(* CoDeSys 2.3.9.48 project: 4.2_EOT20170112.pro *)
(* Libraries: SYSLIBMEM.LIB 8.11.10 18:37:48, C:\Program Files (x86)\WAGO Software\CoDeSys V2.3\Targets\WAGO\Libraries\Application\WagoLibMBX_System_01.lib 22.10.13 22:28:54, C:\Program Files (x86)\WAGO Software\CoDeSys V2.3\Targets\WAGO\Libraries\Application\WagoLibMBX_01.lib 20.3.12 22:32:38, C:\Program Files (x86)\WAGO Software\CoDeSys V2.3\Targets\WAGO\Libraries\Application\WagoLib_CAN_Gateway_02.lib 25.11.15 18:32:40, Util.lib 26.9.14 10:12:46, Standard.lib 8.11.10 18:37:48, SYSLIBCALLBACK.LIB 8.11.10 18:37:48, WagoLibModbus_IP_01.lib 12.2.16 17:20:24, SysLibSockets.lib 5.5.11 15:22:24, WagoLibSockets.lib 14.5.12 18:49:54, NETVARUDP_LIB_V23.LIB 8.11.10 18:37:48, Wago_MBCFG_ETHERNET_01.lib 1.4.15 20:24:28, Wago_MBCFG_COMMON_01.lib 1.4.15 20:24:28 *)

(* PLC configuration (modules and I/O channels)
0753-0430 8 DI 24 V DC 3.0ms [Type_1_8_Channels] node 0, in %IB12 out %QB24 {INTTypePAAssignment = PLC; INTTypeModule = plugged}
  AT %IX6.0 [BOOLOnX_I] Ch_1 Digital input
  AT %IX6.1 [BOOLOnX_I] Ch_2 Digital input
  AT %IX6.2 [BOOLOnX_I] Ch_3 Digital input
  AT %IX6.3 [BOOLOnX_I] Ch_4 Digital input
  AT %IX6.4 [BOOLOnX_I] Ch_5 Digital input
  AT %IX6.5 [BOOLOnX_I] Ch_6 Digital input
  AT %IX6.6 [BOOLOnX_I] Ch_7 Digital input
  AT %IX6.7 [BOOLOnX_I] Ch_8 Digital input
0753-0430 8 DI 24 V DC 3.0ms [Type_1_8_Channels] node 1, in %IB12 out %QB24 {INTTypePAAssignment = PLC; INTTypeModule = plugged}
  AT %IX6.8 [BOOLOnX_I] Ch_1 Digital input
  AT %IX6.9 [BOOLOnX_I] Ch_2 Digital input
  AT %IX6.10 [BOOLOnX_I] Ch_3 Digital input
  AT %IX6.11 [BOOLOnX_I] Ch_4 Digital input
  AT %IX6.12 [BOOLOnX_I] Ch_5 Digital input
  AT %IX6.13 [BOOLOnX_I] Ch_6 Digital input
  AT %IX6.14 [BOOLOnX_I] Ch_7 Digital input
  AT %IX6.15 [BOOLOnX_I] Ch_8 Digital input
0753-0430 8 DI 24 V DC 3.0ms [Type_1_8_Channels] node 2, in %IB13 out %QB24 {INTTypePAAssignment = PLC; INTTypeModule = plugged}
  AT %IX7.0 [BOOLOnX_I] Ch_1 Digital input
  AT %IX7.1 [BOOLOnX_I] Ch_2 Digital input
  AT %IX7.2 [BOOLOnX_I] Ch_3 Digital input
  AT %IX7.3 [BOOLOnX_I] Ch_4 Digital input
  AT %IX7.4 [BOOLOnX_I] Ch_5 Digital input
  AT %IX7.5 [BOOLOnX_I] Ch_6 Digital input
  AT %IX7.6 [BOOLOnX_I] Ch_7 Digital input
  AT %IX7.7 [BOOLOnX_I] Ch_8 Digital input
AT %QX12.0 [BOOLOnX_Q] Ch_1 Digital output
AT %QX12.1 [BOOLOnX_Q] Ch_2 Digital output
AT %QX12.2 [BOOLOnX_Q] Ch_3 Digital output
AT %QX12.3 [BOOLOnX_Q] Ch_4 Digital output
AT %QX12.4 [BOOLOnX_Q] Ch_5 Digital output
AT %QX12.5 [BOOLOnX_Q] Ch_6 Digital output
AT %QX12.6 [BOOLOnX_Q] Ch_7 Digital output
AT %QX12.7 [BOOLOnX_Q] Ch_8 Digital output
AT %QX12.8 [BOOLOnX_Q] Ch_1 Digital output
AT %QX12.9 [BOOLOnX_Q] Ch_2 Digital output
AT %QX12.10 [BOOLOnX_Q] Ch_3 Digital output
AT %QX12.11 [BOOLOnX_Q] Ch_4 Digital output
AT %QX12.12 [BOOLOnX_Q] Ch_5 Digital output
AT %QX12.13 [BOOLOnX_Q] Ch_6 Digital output
AT %QX12.14 [BOOLOnX_Q] Ch_7 Digital output
AT %QX12.15 [BOOLOnX_Q] Ch_8 Digital output
AT %QX13.0 [BOOLOnX_Q] Ch_1 Digital output
AT %QX13.1 [BOOLOnX_Q] Ch_2 Digital output
AT %QX13.2 [BOOLOnX_Q] Ch_3 Digital output
AT %QX13.3 [BOOLOnX_Q] Ch_4 Digital output
AT %QX13.4 [BOOLOnX_Q] Ch_5 Digital output
AT %QX13.5 [BOOLOnX_Q] Ch_6 Digital output
AT %QX13.6 [BOOLOnX_Q] Ch_7 Digital output
AT %QX13.7 [BOOLOnX_Q] Ch_8 Digital output
AT %QW0 [WORDOnW_Q] Ch_1 Analog output
AT %QW1 [WORDOnW_Q] Ch_2 Analog output
AT %QW2 [WORDOnW_Q] Ch_3 Analog output
AT %QW3 [WORDOnW_Q] Ch_4 Analog output
AT %QW4 [WORDOnW_Q] Ch_1 Analog output
AT %QW5 [WORDOnW_Q] Ch_2 Analog output
AT %QW6 [WORDOnW_Q] Ch_3 Analog output
AT %QW7 [WORDOnW_Q] Ch_4 Analog output
AT %IW0 [WORDOnW_I] Ch_1 Input word
AT %IW1 [WORDOnW_I] Ch_2 Input word
AT %IW2 [WORDOnW_I] Ch_1 Input word
AT %IW3 [WORDOnW_I] Ch_2 Input word
AT %IW4 [WORDOnW_I] Ch_1 Input word
AT %IW5 [WORDOnW_I] Ch_2 Input word
0753-0555 4 AO 4-20mA [Type_14_4_Channels] node 6, in %IB20 out %QB32 {INTTypePAAssignment = PLC; INTTypeModule = plugged}
  AT %QW8 [WORDOnW_Q] Ch_1 Analog output
  AT %QW9 [WORDOnW_Q] Ch_2 Analog output
  AT %QW10 [WORDOnW_Q] Ch_3 Analog output
  AT %QW11 [WORDOnW_Q] Ch_4 Analog output
Fieldbus variables [FB_VARS] node 1, in %IB0 out %QB0
Flag variables [FLAG_VARS] node 2, in %IB0 out %QB0
Modbus-Master [MB_MASTER] node 3, in %IB0 out %QB0
*)

(* Global variable list: Global_Variables *)
VAR_GLOBAL

	(*---------------------Control transfer between WING EOT and BRG CENR EOT---------------------*)
	(*control flag*)
	(*control in bridge*)
	BRG_IN_CONTROL_P: BOOL;

	BRG_CENR_IN_CONTROL: BOOL := TRUE;
	BRG_PORT_IN_CONTROL: BOOL := FALSE;
	BRG_STBD_IN_CONTROL: BOOL := FALSE;

	(*during control transfer process flag*)
	CONTROL_TRANS_PROCESS_FLAG: BOOL := FALSE;

	(*EOT LAMP*)
	BRIDGE_PORT_EOT_IN_CONTROL_LAMP: BOOL;
	BRIDGE_STBD_EOT_IN_CONTROL_LAMP: BOOL;
	PORT_EOT_IN_CONTROL_LAMP: BOOL;
	STBD_EOT_IN_CONTROL_LAMP: BOOL;

	(*EOT MVL*)
	PORT_WING_EOT_MVL: WORD;
	CENT_EOT_MVL: WORD;
	STBD_WING_EOT_MVL: WORD;

	(*BUZZER EOT*)
	BRIDGE_BUZZER: BOOL;
	PORT_BUZZER: BOOL;
	STBD_BUZZER: BOOL;


	(*TAKE and SUPPLY button*)
	(*CNTR BUTTON*)
	PORT_BUTTON_EOT_IN_CNTR: BOOL;
	STBD_BUTTON_EOT_IN_CNTR: BOOL;
	(*STBD,PORT  BUTTON*)
	STBD_BUTTON_EOT: BOOL;
	PORT_BUTTON_EOT: BOOL;

	(*Flasher_frequency*)
	Flasher_frequency_P: REAL;


	(*---------------------4.1.7.1.1  MVL Command--------------------*)
	(*input*)
	TELEGRAPH_POSITION_BR: WORD;
	TELEGRAPH_POSITION_CR: WORD;
	TELEGRAPH_POSITION_LC: WORD;

	ECR_AUT_CTRL: BOOL;
	LOCAL_MAN_CTRL: BOOL;
	(*output*)
	TELEGRAPH_INDICATOR_BR: WORD;
	TELEGRAPH_INDICATOR_BR_PORT: WORD;
	TELEGRAPH_INDICATOR_BR_STBD: WORD;
	TELEGRAPH_INDICATOR_ECR: WORD;
	TELEGRAPH_INDICATOR_LC: WORD;

	(**************MVL POWER LOST**************)
	(*INPUT*)
	ECR_TElegraph_POWER_LOST_P: BOOL;
	LOCAL_TElegraph_POWER_LOST_P: BOOL;
	PORT_TElegraph_POWER_LOST_P: BOOL;
	STBD_TElegraph_POWER_LOST_P: BOOL;
	BR_TElegraph_POWER_LOST_P: BOOL;

	TELEGRAPH_SUB_SYS_PWR_LOST: BOOL;



	(*---------------------4.1.7.1.2  Sub-telegraph function--------------------*)
	(*current status
	0 = NOSTATUS; 1 = STANDBY; 2 = AT SEA; 3 = FWE*)
	AUX_EOT_STATUS: UDINT := 0;

	(*PUSHBUTTON*)
	PUSHBUTTON_STANDBY_BRG: BOOL;
	PUSHBUTTON_ATSEA_BRG: BOOL;
	PUSHBUTTON_FWE_BRG: BOOL;

	PUSHBUTTON_STANDBY_MCR: BOOL;
	PUSHBUTTON_ATSEA_MCR: BOOL;
	PUSHBUTTON_FWE_MCR: BOOL;

	(*indicator*)
	INDICATOR_STANDBY_BRG: BOOL;
	INDICATOR_ATSEA_BRG: BOOL;
	INDICATOR_FWE_BRG: BOOL;

	INDICATOR_STANDBY_MCR: BOOL;
	INDICATOR_ATSEA_MCR: BOOL;
	INDICATOR_FWE_MCR: BOOL;

	INDICATOR_STANDBY_LC: BOOL;
	INDICATOR_ATSEA_LC: BOOL;
	INDICATOR_FWE_LC: BOOL;

	(*buzzers, FALSE = silence; TRUE = activated*)
	BUZZER_BRG: BOOL;
	BUZZER_MCR: BOOL;

	(*Is during switch process NO = FALSE; YES = TRUE*)
	MODE_TRANSFER_FLAG: BOOL := FALSE;

	H_AT_SEA: BOOL; (*PROEOT0003*)
	H_STAND_BY: BOOL;(*PROEOT0004*)
	H_FINSHED_WITH_ENGINE: BOOL;(*PROEOT0005*)


	(*---------------------4.1.7.1.3  Wrong way--------------------*)
	(*input*)
	MVL_POSITION_AHEAD: BOOL;
	MVL_POSITION_ASTERN: BOOL;
	ENGINE_TURN_AHEAD: BOOL;
	ENGINE_TURN_ASTERN: BOOL;
	MCR_LC_CONTROL: BOOL;
	ECR_MAN_CONTROL: BOOL;

	(*output*)
	WRONG_WAY: BOOL;

	(*---------------------4.1.7.1.4  Mismatch Alarm--------------------*)
	(*input*)
	TELEGRAPH_ORDER_THRESHOLD_INPUT: WORD;(*2ma*)
	(*output*)
	TELEGRAPH_ORDER_BR: BOOL;
	TELEGRAPH_ORDER_PORT: BOOL;
	TELEGRAPH_ORDER_STBD: BOOL;
	TELEGRAPH_ORDER_ECR: BOOL;
	TELEGRAPH_ORDER_LC: BOOL;

	TELEGRAPH_COINCIDENCE: BOOL;

	(*silence  MISMATCH BUZZER*)
	ESS_BR_ALARM_ACK_P:    BOOL;
	ESS_ECR_ALARM_ACK_P:   BOOL;
	ESS_PORT_ALARM_ACK_P:   BOOL;
	ESS_STBD_ALARM_ACK_P:   BOOL;

	(*---------------------4.1.7.1.5  EOT system failure Alarm--------------------*)
	(*input*)
	PASSIVE_FAIL_THRESHOLD: WORD;(*2ma*)
	(*output*)
	PASSIVE_FAILURE_BR: BOOL;
	PASSIVE_FAILURE_BR_PORT: BOOL;
	PASSIVE_FAILURE_BR_STBD: BOOL;
	PASSIVE_FAILURE_ECR: BOOL;
	PASSIVE_FAILURE_LC: BOOL;

	TELEGRAPH_SYSTEM_FAIL_XS9021A: BOOL;

	(*---------------------LAMP TEST PB FROM RCS--------------------*)
	ECR_LAMP_TEST_PB: BOOL;
	BR_LAMP_TEST_PB: BOOL;
	PORT_LAMP_TEST_PB: BOOL;
	STBD_LAMP_TEST_PB: BOOL;

	(*4 lamp test PB OR*)
	LAMP_TEST_PB:	BOOL;
	BRIDGE_LAMP_TEST_PB:	BOOL;

	(*-------------------------------AMPERE STAGE TO HMI-------------------------------*)
	(*750-452  AI 输入模块 0~20mA, 20mA对应32760,  AD_Scale 为32760/20*)
	AD_Scale: WORD := 1638;
	(*750-555  AO 输出模块 4~20mA, 20mA对应32760, DA_Scale 为32760/16*)
	DA_Scale: WORD := 2048;

	AMPERE_STAGE_TO_HMI: WORD;		(*
												   bit 0	Emergency  AS
												   bit 1   FULL.AS
												   bit 2   HALF AS
												   bit 3  	SLOW  AS
												   bit 4   DEAD  S. AH
												   bit 5   STOP
												   bit 6   DEAD  S. AH
												   bit 7   SLOW  AH
												   bit 8   HALF  AH
												   bit 9   FULL  AH 
												   bit 10   Full SEA  AH*)


	(*LEVEL	INDICATOR*)
	Telegraph_Indicator_Full_SEA_AH: BOOL;
	Telegraph_Indicator_FULL_AH: BOOL;
	Telegraph_Indicator_HALF_AH: BOOL;
	Telegraph_Indicator_SLOW_AH: BOOL;
	Telegraph_Indicator_DEAD_S_AH: BOOL;
	Telegraph_Indicator_STOP: BOOL;
	Telegraph_Indicator_DEAD_S_AS: BOOL;
	Telegraph_Indicator_SLOW_AS: BOOL;
	Telegraph_Indicator_HALF_AS: BOOL;
	Telegraph_Indicator_FULL_AS: BOOL;
	Telegraph_Indicator_Emergency_AS: BOOL;

	(*LEVEL CMD*)
	Telegraph_CMD_Full_SEA_AH: BOOL;
	Telegraph_CMD_FULL_AH: BOOL;
	Telegraph_CMD_HALF_AH: BOOL;
	Telegraph_CMD_SLOW_AH: BOOL;
	Telegraph_CMD_DEAD_S_AH: BOOL;
	Telegraph_CMD_STOP: BOOL;
	Telegraph_CMD_DEAD_S_AS: BOOL;
	Telegraph_CMD_SLOW_AS: BOOL;
	Telegraph_CMD_HALF_AS: BOOL;
	Telegraph_CMD_FULL_AS: BOOL;
	Telegraph_CMD_Emergency_AS: BOOL;

	(***************************MVL_COMMD_TO_AO*******************************)
	BR_MVL_COMMD_TO_RCS_P: WORD;
	ECR_MVL_COMMD_TO_RCS_P: WORD;

	(*INDICATOR OF  BR  MCR  LC*)
	BR_Indicator_Position_Pointer_P:	WORD;
	ECR_Indicator_Position_Pointer_P:  WORD;
	LOCAL_Indicator_Position_Pointer_P:	WORD;

	BR_PORT_Indicator_Position_Pointer_P:	WORD;
	BR_STBD_Indicator_Position_Pointer_P:	WORD;

	(*TEST*)
	TEST_LOCAL_Telegraph_Position_Pointer_P :  WORD;

	(****************************MVL_TO_RCS_TEST_MBS---12.27*******************************)
	BR_MVL_TO_RCS_MBS_P	AT %QW275:	WORD;
	ECR_MVL_TO_RCS_MBS_P		AT %QW277:	WORD;

	BR_MVL_TO_RCS_MBS_P1		AT %QW279:	WORD;
	ECR_MVL_TO_RCS_MBS_P1		AT %QW281:	WORD;


	(***************************EOT HW Signal list*******************************)
	(*-----------AI----------*)
	BR_MVL_COMMD									AT	%IW0: WORD;(*PROEOT1001*)
	ECR_MVL_COMMD								AT	%IW1: WORD;(*PROEOT1002*)
	LOCAL_MVL_COMMD							AT	%IW2: WORD;(*PROEOT1003*)
	PORT_BR_MVL_COMMD: 				WORD;(*PROEOT1004*)
	STBD_BR_MVL_COMMD: 				WORD;(*PROEOT1005*)

	(*-----------AO----------*)
	BR_Indicator_Position_Pointer					AT	%QW0: WORD;(*PROEOT1006*)
	BR_MVL_COMMD_TO_RCS					       AT %QW4: WORD;(*PROEOT1007*)
	ECR_Indicator_Position_Pointer					AT	%QW1: WORD;(*PROEOT1008*)
	ECR_MVL_COMMD_TO_RCS 					AT%QW5: WORD;(*PROEOT1009*)
	LOCAL_Indicator_Position_Pointer				AT	%QW2: WORD;(*PROEOT1010*)
	PORT_BR_Indicator_Position_Pointer: REAL;(*PROEOT1011*)
	STBD_BR_Indicator_Position_Pointer: REAL;(*PROEOT1012*)
	(*TEST*)
	TEST_LOCAL_Telegraph_Position_Pointer		AT	%QW3: WORD;(*PROEOT1010*)

	(*-----------DI----------*)
	STANDBY_BR_PB								AT	%IX6.0: BOOL;(*PROEOT1013*)
	AT_SEA_BR_PB									AT	%IX6.1: BOOL;(*PROEOT1014*)
	FWE_BR_PB										AT	%IX6.2: BOOL;(*PROEOT1015*)
	BR_TElegraph_POWER_LOST					AT	%IX6.3: BOOL;(*PROEOT1016*)
	STANDBY_ECR_AUT_PB						AT	%IX6.4: BOOL;(*PROEOT1017*)
	AT_SEA_ECR_AUT_PB							AT	%IX6.5: BOOL;(*PROEOT1018*)
	FWE_ECR_AUT_PB								AT	%IX6.6: BOOL;(*PROEOT1019*)
	ECR_TElegraph_POWER_LOST				AT	%IX6.7: BOOL;(*PROEOT1020*)
	LOCAL_TElegraph_POWER_LOST				AT	%IX6.10: BOOL;(*PROEOT1021*)
	PORT_TElegraph_POWER_LOST: BOOL;(*PROEOT1022*)
	STBD_TElegraph_POWER_LOST: BOOL;(*PROEOT1023*)
	BR_CENTRL_PORT_APPLY_FOR_CONTROL: BOOL;(*PROEOT1024*)
	BR_CENTRL_STBD_APPLY_FOR_CONTROL: BOOL;(*PROEOT1025*)
	BR_PORT_APPLY_FOR_CONTROL: BOOL;(*PROEOT1026*)
	BR_STBD_APPLY_FOR_CONTROL: BOOL;(*PROEOT1027*)
	LOCAL_IN_CONTROL_TAKE_ON				AT	%IX7.1: BOOL;(*PROEOT1028*)


	(*-----------DO----------*)
	STANDBY_BR_INDICATOR									AT	%QX12.0: BOOL;(*PROEOT1029*)
	AT_SEA_BR_PB_INDICATOR								AT	%QX12.1: BOOL;(*PROEOT1030*)
	FWE_BR_PB_INDICATOR									AT	%QX12.2: BOOL;(*PROEOT1031*)
	BR_TELEGRAPH_ORDER_Acoustic_Signal				AT	%QX12.3: BOOL;(*PROEOT1032*)
	STANDBY_ECR_AUT_PB_INDICATOR						AT	%QX12.4: BOOL;(*PROEOT1033*)
	AT_SEA_ECR_AUT_PB_INDICATOR						AT	%QX12.5: BOOL;(*PROEOT1034*)
	FWE_ECR_AUT_PB_INDICATOR							AT	%QX12.6: BOOL;(*PROEOT1035*)
	ECR_TELEGRAPH_ORDER_Acoustic_Signal				AT	%QX12.7: BOOL;(*PROEOT1036*)
	STANDBY_LOCAL_INDICATOR: BOOL;(*PROEOT1037*)
	AT_SEA_LOCAL_INDICATOR: BOOL;(*PROEOT1038*)
	FWE_LOCAL_INDICATOR: BOOL;(*PROEOT1039*)
	LOCAL_TELEGRAPH_ORDER_Acoustic_Signal			AT	%QX12.10: BOOL;(*PROEOT1040*)
	PORT_TELEGRAPH_ORDER_Acoustic_Signal: BOOL;(*PROEOT1041*)
	STBD_TELEGRAPH_ORDER_Acoustic_Signal: BOOL;(*PROEOT1042*)
	BR_CENTRL_PORT_CONTROL_IN_CONTROL: BOOL;(*PROEOT1043*)
	BR_CENTRL_STBD_CONTROL_IN_CONTROL: BOOL;(*PROEOT1044*)
	BR_PORT_CONTROL_IN_CONTROL: BOOL;(*PROEOT1045*)
	BR_STBD_CONTROL_IN_CONTROL: BOOL;(*PROEOT1046*)
	LOCAL_IN_CONTROL_TAKE_ON_INDICATOR				AT	%QX13.1: BOOL;(*PROEOT1047*)
	Telegraph_System_Failure_ALM								AT	%QX13.2: BOOL;(*PROEOTXS9021A*)
	HW_WRONG_WAY_BR										AT	%QX13.3:  BOOL;
	HW_WRONG_WAY_ECR										AT	%QX13.4:  BOOL;
	HW_WRONG_WAY_LC										AT	%QX13.5:  BOOL;

	(*PORT or STBD in control *)
	HW_PORT_IN_CONTROL: BOOL;	(*PROEOT1048*)
	HW_STBD_IN_CONTROL: BOOL;	(*PROEOT1049*)


	(****************************EOT & HMI COMMUNICATION SIGNALS LIST*******************************)
	(*STRING*)

  	SWD_swd_ctr_mode_0 AT %QW271: UINT;


	(*SDO*)

	LOCAL_MAN_TAKE_OVER   AT	%QX260.11: BOOL;(*PROEOT0019       SP_swd_perm_eot1_12_62*)
	H_PORT_WING_CONTRL  AT	%QX260.12: BOOL;(*PROEOT0025       SP_swd_perm_eot1_13_62*)
	H_STBD_WING_CONTRL   AT	%QX259.13: BOOL;(*PROEOT0026    SP_swd_perm_eot1_14_62*)

	H_BR_TElegraph_POWER_LOST  AT	%QX261.0: BOOL;(*PROEOT0029    SP_swd_perm_eot2_1_62*)
	H_ECR_TElegraph_POWER_LOST  AT	%QX261.1: BOOL;(*PROEOT0030   SP_swd_perm_eot2_2_62*)
	H_LOCAL_TElegraph_POWER_LOST  AT	%QX261.2: BOOL;(*PROEOT0031   SP_swd_perm_eot2_3_62*)
	H_PORT_TElegraph_POWER_LOST  AT	%QX261.3: BOOL;(*PROEOT0032    SP_swd_perm_eot2_4_62*)
	H_STBD_TElegraph_POWER_LOST  AT	%QX261.4: BOOL;(*PROEOT0033   SP_swd_perm_eot2_5_62*)

	H_BR_TElegraph_PASSIVE_FAIL  AT	%QX261.5: BOOL;(*PROEOT0034  SP_swd_perm_eot2_6_62*)
	H_ECR_TElegraph_PASSIVE_FAIL  AT	%QX261.6: BOOL;(*PROEOT0035   SP_swd_perm_eot2_7_62*)
	H_LOCAL_TElegraph_PASSIVE_FAIL  AT	%QX261.7: BOOL;(*PROEOT0036   SP_swd_perm_eot2_8_62*)
	H_PORT_TElegraph_PASSIVE_FAIL  AT	%QX261.8: BOOL;(*PROEOT0037    SP_swd_perm_eot2_9_62*)
	H_STBD_TElegraph_PASSIVE_FAIL  AT	%QX261.9: BOOL;(*PROEOT0038   SP_swd_perm_eot2_10_62*)

	TELEGRAPH_HORN_ALARM_MBO   AT   %QX261.10: BOOL;   (*PROEOT0039   SP_swd_perm_eot2_11_62*)
	TELEGRAPH_SUB_SYS_PWR_LOST_MBO   AT   %QX261.11: BOOL;   (*PROEOT0044   SP_swd_perm_eot2_12_62*)
	TELEGRAPH_SYS_PASS_FAIL_9021A_MBO   AT   %QX261.12: BOOL;  (*PROEOTXS9021A   SP_swd_perm_eot2_13_62*)

	H_TELEGRAPH_COINCIDENCE   AT   %QX261.13: BOOL;  (*PROEOT9001  SP_swd_perm_eot2_14_62*)
	H_WRONG_WAY	 AT   %QX261.14:  BOOL; 	(*PROEOT9050  SP_swd_perm_eot2_15_62*)

	(*Corresponding  Ampere to  HMI-----------------------New Signal*)
	Telegraph_Indicator_Full_SEA_AH_MBO      AT  %QX260.0: BOOL;  (*PROEOT0001      SP_swd_perm_eot1_1_62 *)
	Telegraph_Indicator_FULL_AH_MBO      AT  %QX260.1: BOOL;  (*PROEOT0002      SP_swd_perm_eot1_2_62 *)
	Telegraph_Indicator_HALF_AH_MBO      AT  %QX260.2: BOOL;  (*PROEOT0003      SP_swd_perm_eot1_3_62 *)
	Telegraph_Indicator_SLOW_AH_MBO      AT  %QX260.3: BOOL;  (*PROEOT0004      SP_swd_perm_eot1_4_62 *)
	Telegraph_Indicator_DEAD_S_AH_MBO      AT  %QX260.4: BOOL;  (*PROEOT0005      SP_swd_perm_eot1_5_62 *)
	Telegraph_Indicator_STOP_MBO      AT  %QX260.5: BOOL;  (*PROEOT0006      SP_swd_perm_eot1_6_62 *)
	Telegraph_Indicator_DEAD_S_AS_MBO      AT  %QX260.6: BOOL;  (*PROEOT0007      SP_swd_perm_eot1_7_62 *)
	Telegraph_Indicator_SLOW_AS_MBO      AT  %QX260.7: BOOL;  (*PROEOT0008      SP_swd_perm_eot1_8_62 *)
	Telegraph_Indicator_HALF_AS_MBO      AT  %QX260.8: BOOL;  (*PROEOT0009      SP_swd_perm_eot1_9_62 *)
	Telegraph_Indicator_FULL_AS_MBO      AT  %QX260.9: BOOL;  (*PROEOT0010      SP_swd_perm_eot1_10_62 *)
	Telegraph_Indicator_Emergency_AS_MBO      AT  %QX260.10: BOOL;  (*PROEOT0011      SP_swd_perm_eot1_11_62 *)


	(****************************RCS TO EOT 		ESS TO EOT   MODBUS  COMMUNICATION SIGNALS LIST*******************************)
(*	FRM_BR_CONTROL     AT  %IX262.0: BOOL;    (*PROEOT0017      SP_swd_perm_eotout_1_62  *)
	FRM_ECR_AUT_CONTROL     AT  %IX262.1: BOOL;    (*PROEOT0018      SP_swd_perm_eotout_2_62  *)
	FRM_ECR_LAMP_TEST_PB     AT  %IX262.2: BOOL;    (*PROEOT0040      SP_swd_perm_eotout_3_62  *)
	FRM_BR_LAMP_TEST_PB     AT  %IX262.3: BOOL;    (*PROEOT0041      SP_swd_perm_eotout_4_62  *)
	FRM_PORT_LAMP_TEST_PB     AT  %IX262.4: BOOL;    (*PROEOT0042      SP_swd_perm_eotout_5_62  *)
	FRM_STBD_LAMP_TEST_PB     AT  %IX262.5: BOOL;    (*PROEOT0043      SP_swd_perm_eotout_6_62  *)


	ESS_BR_ALARM_ACK     AT  %IX262.6: BOOL;    (*PROEOT0045	SP_swd_perm_eotout_7_62  *)
	ESS_ECR_ALARM_ACK     AT  %IX262.7: BOOL;    (*PROEOT0046	SP_swd_perm_eotout_8_62  *)
	ESS_PORT_ALARM_ACK     AT  %IX262.8: BOOL;    (*PROEOT0047	SP_swd_perm_eotout_9_62  *)
	ESS_STBD_ALARM_ACK     AT  %IX262.9: BOOL;    (*PROEOT0048	SP_swd_perm_eotout_10_62  *)  CXJ   2016-12-21*)

	FRM_BR_CONTROL  : BOOL;    (*PROEOT0017    PRORCCAN2001      SP_swd_perm_eotout_1_62  *)
	FRM_ECR_AUT_CONTROL  : BOOL;    (*PROEOT0018     PRORCCAN2002    SP_swd_perm_eotout_2_62  *)
	FRM_ECR_LAMP_TEST_PB  : BOOL;    (*PROEOT0040    PRORCS0139      SP_swd_perm_eotout_3_62  *)
	FRM_BR_LAMP_TEST_PB  : BOOL;    (*PROEOT0041       PRORCS0140   SP_swd_perm_eotout_4_62  *)
	FRM_PORT_LAMP_TEST_PB   : BOOL;    (*PROEOT0042     PRORCS0141   SP_swd_perm_eotout_5_62  *)
	FRM_STBD_LAMP_TEST_PB   : BOOL;    (*PROEOT0043      PRORCS0142   SP_swd_perm_eotout_6_62  *)
	FRM_ECR_MAN_CONTROL  : BOOL;
	FRM_LOCAL_MAN_CONTROL  : BOOL;
	FRM_CONTROL_TRANS_BUZZER_BRG :BOOL;
	FRM_CONTROL_TRANS_BUZZER_MCR:BOOL;
	FRM_FAIL_ACOUSTIC_BUZZER:BOOL;

	ESS_BR_ALARM_ACK   : BOOL;    (*PROEOT0045	 PROESS0118  SP_swd_perm_eotout_7_62  *)
	ESS_ECR_ALARM_ACK   : BOOL;    (*PROEOT0046   PROESS0119  	SP_swd_perm_eotout_8_62  *)
	ESS_PORT_ALARM_ACK   : BOOL;    (*PROEOT0047	 PROESS0120   SP_swd_perm_eotout_9_62  *)
	ESS_STBD_ALARM_ACK   : BOOL;    (*PROEOT0048	PROESS0121   SP_swd_perm_eotout_10_62  *)

	(*ENG STATUS FROM RCS AND ESS*)
	FRM_ENG_TURNING_AHEAD:BOOL;
	FRM_ENG_TURNING_AST:BOOL;
	FRM_ENG_SENSOR_1_FAILURE:BOOL;

	ESS_ENG_TURNING_AHEAD:BOOL;
	ESS_ENG_TURNING_AST:BOOL;
	ESS_ENG_SENSOR_1_FAILURE:BOOL;

END_VAR


VAR_GLOBAL RETAIN
	(*Set  Point*)
	SPT_tlg_order_thld   AT   %IW258:  REAL := 2;  (*1ma = 1024*) (*PROEOT0001*)
	SPT_tlg_flasher_freq  AT	%IW256:  REAL := 1; (*default 1hz *)(*PROEOT0002*)
END_VAR

(* Global variable list: Networkmanagement implicit Variables UDP *)
VAR_GLOBAL CONSTANT
	USE_NWVARS_UDP : BOOL := FALSE;
	MAX_NetVarItems_UDP	: INT := 0;
	MAX_NetVarPDO_Rx_UDP	: INT := 0;
	MAX_NetVarPDO_Tx_UDP	: INT := 0;
	MAX_NetVarOD_UDP		: INT := 0;
END_VAR
VAR_GLOBAL
	pNetVarItems_UDP		: ARRAY[0..MAX_NetVarItems_UDP] OF NetVarDataItem_UDP;
	pNetVarPDO_Rx_UDP		: ARRAY[0..MAX_NetVarPDO_Rx_UDP] OF NetVarPDO_Rx_UDP;
	pNetVarPDO_Tx_UDP		: ARRAY[0..MAX_NetVarPDO_Tx_UDP] OF NetVarPDO_Tx_UDP;
	pNetVarOD_UDP			: ARRAY[0..MAX_NetVarOD_UDP] OF NetVarSDO_UDP;
	pNetVarPDO_Rx_Diagnosis_UDP : ARRAY[0..MAX_NetVarPDO_Rx_UDP] OF NetVarUDPDiagStruct;
	pNetVarPDO_Tx_Diagnosis_UDP : ARRAY[0..MAX_NetVarPDO_Tx_UDP] OF NetVarUDPDiagStruct;
END_VAR

(* POU PLC_PRG, ST *)
PROGRAM PLC_PRG
VAR
	(**********FUNCTION BLOCK**************)
	InputProgramValueMapping_FUNC: InputProgramValueMapping;
	SWD_FUNC: SWD;
	OutputProgramValueMapping_FUNC: OutputProgramValueMapping;
	MVL_COMMAND_FUNC: MVL_COMMAND;
	Sub_telegraph_function_FUNC: Sub_telegraph_function;
	WRONG_WAY_FUNC: WRONG_WAY;
	MISMATCH_ALARM_FUNC: MISMATCH_ALARM;
	EOT_system_failure_Alarm_FUNC: EOT_system_failure_Alarm;
	LAMP_TEST_FUNC: LAMP_TEST;
	AMPERE_STAGE_TO_HMI_FUNC: AMPERE_STAGE_TO_HMI;
	MVL_COMMD_TO_AO_FUNC: MVL_COMMD_TO_AO;
	(*TEST 12.27*)
	MVL_TO_RCS_TEST_MBS_FUNC:	MVL_TO_RCS_TEST_MBS;
	Bridge_Control_Position_Change_FUNC: Bridge_Control_Position_Change;
END_VAR
(*************************Input  Program Value Mapping**********************************)
InputProgramValueMapping_FUNC;


(*************************SWD_FUNC**********************************)
SWD_FUNC;

(*************************Bridge_Control_Position_Change**********************************)
Bridge_Control_Position_Change_FUNC;


(*************************MVL_COMMAND**********************************)
MVL_COMMAND_FUNC;


(*************************AMPERE_STAGE_TO_HMI**********************************)
AMPERE_STAGE_TO_HMI_FUNC;


(*************************Sub_telegraph_function**********************************)
Sub_telegraph_function_FUNC;


(*************************WRONG_WAY**********************************)
WRONG_WAY_FUNC;


(*************************MISMATCH_ALARM**********************************)
MISMATCH_ALARM_FUNC;


(*************************EOT_system_failure_Alarm**********************************)
EOT_system_failure_Alarm_FUNC;


(*************************MVL_COMMD_TO_AO**********************************)
(*convert  AI  to  AO*)
MVL_COMMD_TO_AO_FUNC;


(*************************LAMP  TEST  PROCESS**********************************)
(*     NO'T USED
LAMP_TEST_FUNC;
*)

(*************************Output  Program Value Mapping**********************************)
OutputProgramValueMapping_FUNC;


(**********************TEST MVL CMD TO RCS FROM MBS*****************************)
MVL_TO_RCS_TEST_MBS_FUNC;
END_PROGRAM

(* POU InputProgramValueMapping, ST *)
FUNCTION_BLOCK InputProgramValueMapping
VAR_INPUT
END_VAR
VAR_OUTPUT
END_VAR
VAR
END_VAR
(*****该函数块用于获取所有程序外部输入变量并赋值给程序定义的内部全局变量,包括setpoint, HW input, MODBUS input*****)

(*CXJ----2016-12-21*)
	(*Modbus  input*)
     MODBUS_CONFIGURATION;
      IF  MBCFG_RCS.MBCFG_Error=MBCFG_NO_ERROR  THEN
	FRM_BR_CONTROL  :=MBCFG_RCS.FRM_BR_CONTROL_cfg    ;    (*PROEOT0017    PRORCCAN2001      SP_swd_perm_eotout_1_62  *)
	FRM_ECR_AUT_CONTROL  :=MBCFG_RCS.FRM_ECR_AUT_CONTROL_cfg   ;    (*PROEOT0018     PRORCCAN2002    SP_swd_perm_eotout_2_62  *)
	FRM_ECR_LAMP_TEST_PB  :=MBCFG_RCS.FRM_ECR_LAMP_TEST_PB_cfg   ;    (*PROEOT0040    PRORCS0139      SP_swd_perm_eotout_3_62  *)
	FRM_BR_LAMP_TEST_PB  :=MBCFG_RCS.FRM_BR_LAMP_TEST_PB_cfg  ;    (*PROEOT0041       PRORCS0140   SP_swd_perm_eotout_4_62  *)
	FRM_PORT_LAMP_TEST_PB   :=MBCFG_RCS.FRM_PORT_LAMP_TEST_PB_cfg;    (*PROEOT0042     PRORCS0141   SP_swd_perm_eotout_5_62  *)
	FRM_STBD_LAMP_TEST_PB   :=MBCFG_RCS.FRM_STBD_LAMP_TEST_PB_cfg;    (*PROEOT0043      PRORCS0142   SP_swd_perm_eotout_6_62  *)
	FRM_ECR_MAN_CONTROL := MBCFG_RCS.FRM_ECR_MAN_CONTROL_cfg;
	FRM_LOCAL_MAN_CONTROL  :=  MBCFG_RCS.FRM_LOCAL_MAN_CONTROL_cfg;
	FRM_FAIL_ACOUSTIC_BUZZER :=MBCFG_RCS.FRM_FAIL_ACOUSTIC_cfg;
	FRM_CONTROL_TRANS_BUZZER_BRG:=MBCFG_RCS.FRM_CONTROL_TRANS_BUZZER_BRG_cfg;
	FRM_CONTROL_TRANS_BUZZER_MCR:=MBCFG_RCS.FRM_CONTROL_TRANS_BUZZER_MCR_cfg;

	FRM_ENG_TURNING_AHEAD:= MBCFG_RCS.FRM_ENG_TURNING_AHEAD_cfg;
	FRM_ENG_TURNING_AST := MBCFG_RCS.FRM_ENG_TURNING_AST_cfg;
	FRM_ENG_SENSOR_1_FAILURE := MBCFG_RCS.FRM_ENG_SENSOR_1_FAILURE_cfg;
       END_IF;

       IF MBCFG_ESS.MBCFG_Error=MBCFG_NO_ERROR  THEN
	ESS_BR_ALARM_ACK   :=MBCFG_ESS.ESS_BR_ALARM_ACK_cfg;    (*PROEOT0045	 PROESS0118  SP_swd_perm_eotout_7_62  *)
	ESS_ECR_ALARM_ACK   :=MBCFG_ESS.ESS_ECR_ALARM_ACK_cfg;    (*PROEOT0046   PROESS0119  	SP_swd_perm_eotout_8_62  *)
	ESS_PORT_ALARM_ACK   :=MBCFG_ESS.ESS_PORT_ALARM_ACK_cfg;    (*PROEOT0047	 PROESS0120   SP_swd_perm_eotout_9_62  *)
	ESS_STBD_ALARM_ACK   :=MBCFG_ESS.ESS_STBD_ALARM_ACK_cfg;    (*PROEOT0048	PROESS0121   SP_swd_perm_eotout_10_62  *)

	ESS_ENG_TURNING_AHEAD := MBCFG_ESS.ESS_ENG_TURNING_AHEAD_cfg;
	ESS_ENG_TURNING_AST := MBCFG_ESS.ESS_ENG_TURNING_AST_cfg;
	ESS_ENG_SENSOR_1_FAILURE := MBCFG_ESS.ESS_ENG_SENSOR_1_FAILURE_cfg;
       END_IF;


(***************Bridge_Control_Position_Change***************)
CENT_EOT_MVL := BR_MVL_COMMD;(*PROEOT1001*)
PORT_WING_EOT_MVL := PORT_BR_MVL_COMMD;(*PROEOT1004*)
STBD_WING_EOT_MVL := STBD_BR_MVL_COMMD;(*PROEOT1005*)

BRG_IN_CONTROL_P := FRM_BR_CONTROL;   (*PRORCS0143*)

(***TAKE and SUPPLY button***)
(***CNTR BUTTON***)
PORT_BUTTON_EOT_IN_CNTR := BR_CENTRL_PORT_APPLY_FOR_CONTROL;(*PROEOT1024*)
STBD_BUTTON_EOT_IN_CNTR := BR_CENTRL_STBD_APPLY_FOR_CONTROL;(*PROEOT1025*)
(***STBD,PORT  BUTTON***)
PORT_BUTTON_EOT := BR_PORT_APPLY_FOR_CONTROL;(*PROEOT1026*)
STBD_BUTTON_EOT := BR_STBD_APPLY_FOR_CONTROL;(*PROEOT1027*)

(*Flasher_frequency*)
Flasher_frequency_P :=  SPT_tlg_flasher_freq;

(***************MVL COMMAND***************)
TELEGRAPH_POSITION_CR := ECR_MVL_COMMD;(*PROEOT1002*)
TELEGRAPH_POSITION_LC := LOCAL_MVL_COMMD;(*PROEOT1003*)
ECR_AUT_CTRL := FRM_ECR_AUT_CONTROL;  (*PRORCS0144*)
LOCAL_MAN_CTRL := LOCAL_IN_CONTROL_TAKE_ON
						OR  FRM_LOCAL_MAN_CONTROL;(*PROEOT1028*)

(*MVL POWER LOST*)
ECR_TElegraph_POWER_LOST_P := ECR_TElegraph_POWER_LOST; (*PROEOT1020*)
LOCAL_TElegraph_POWER_LOST_P := LOCAL_TElegraph_POWER_LOST; (*PROEOT1021*)
PORT_TElegraph_POWER_LOST_P := PORT_TElegraph_POWER_LOST; (*PROEOT1022*)
STBD_TElegraph_POWER_LOST_P := STBD_TElegraph_POWER_LOST; (*PROEOT1023*)
BR_TElegraph_POWER_LOST_P := BR_TElegraph_POWER_LOST; (*PROEOT1016*)


(***************Sub_telegraph_function***************)
(*PUSHBUTTON*)
PUSHBUTTON_STANDBY_BRG := STANDBY_BR_PB;(*PROEOT1013*)
PUSHBUTTON_ATSEA_BRG := AT_SEA_BR_PB;(*PROEOT1014*)
PUSHBUTTON_FWE_BRG := FWE_BR_PB;(*PROEOT1015*)

PUSHBUTTON_STANDBY_MCR := STANDBY_ECR_AUT_PB;(*PROEOT1017*)
PUSHBUTTON_ATSEA_MCR := AT_SEA_ECR_AUT_PB;(*PROEOT1018*)
PUSHBUTTON_FWE_MCR := FWE_ECR_AUT_PB;(*PROEOT1019*)

(***************Wrong  Way***************)
ECR_MAN_CONTROL := FRM_ECR_MAN_CONTROL;


(***************Mismatch Alarm***************)
(*TELEGRAPH_ORDER_THRESHOLD_INPUT := SPT_tlg_order_thld * AD_Scale;*)

ESS_BR_ALARM_ACK_P := ESS_BR_ALARM_ACK;
ESS_ECR_ALARM_ACK_P := ESS_ECR_ALARM_ACK;
ESS_PORT_ALARM_ACK_P := ESS_PORT_ALARM_ACK;
ESS_STBD_ALARM_ACK_P := ESS_STBD_ALARM_ACK;


(***************LAMP  TEST***************)
ECR_LAMP_TEST_PB := FRM_ECR_LAMP_TEST_PB;  (*PRORCS0139*)
BR_LAMP_TEST_PB := FRM_BR_LAMP_TEST_PB;   (*PRORCS0140*)
PORT_LAMP_TEST_PB := FRM_PORT_LAMP_TEST_PB;   (*PRORCS0141*)
STBD_LAMP_TEST_PB := FRM_STBD_LAMP_TEST_PB;    (*PRORCS0142*)

LAMP_TEST_PB	:=	ECR_LAMP_TEST_PB
					OR	BR_LAMP_TEST_PB
					OR	PORT_LAMP_TEST_PB
					OR	STBD_LAMP_TEST_PB;

BRIDGE_LAMP_TEST_PB :=	BR_LAMP_TEST_PB
							OR	PORT_LAMP_TEST_PB
							OR	STBD_LAMP_TEST_PB;
END_FUNCTION_BLOCK

(* POU Configuration/MODBUS_CONFIGURATION, ST *)
PROGRAM MODBUS_CONFIGURATION        
VAR                                
END_VAR                            
(*                                 
   <?xml version="1.0" encoding="UTF-16" standalone="yes"?>
<network xml_structure_version="1" xml_feature_version="1">
	<generator_settings minRTUTaskCycleTimeMs="5" minEthaskCycleTimeMs="5" ethSlaveMultiplier="0.1" rtuInterfaceMultiplier="0.1" taskGeneration="false"/>
	<master_interface type="eth" name="" expanded="true">
		<mb_slave comment="Ethernet MR Controller 100MBit 2Port" name="RCS" expanded="true" type="wago" article-no="0750-0882">
			<mb_connection type="eth" transport="TCP" port="502" ip="192.168.1.1" unitid="1" request_delay_ms="0" response_timeout_ms="20"/>
			<service_connection type="eth" ip="192.168.1.1"/>
			<generic_vars comment="" expanded="false"/>
			<pfc_vars comment="" expanded="true">
				<pfc_var name="FRM_BR_CONTROL_cfg" comment="" data_type="BOOL" iec_addr="%QX285.0" expanded="false" mb_access="ro" explicitAccess="false"/>
				<pfc_var name="FRM_ECR_AUT_CONTROL_cfg" comment="" data_type="BOOL" iec_addr="%QX285.1" expanded="false" mb_access="ro" explicitAccess="false"/>
				<pfc_var name="FRM_ECR_LAMP_TEST_PB_cfg" comment="" data_type="BOOL" iec_addr="%QX288.9" expanded="false" mb_access="ro" explicitAccess="false"/>
				<pfc_var name="FRM_BR_LAMP_TEST_PB_cfg" comment="" data_type="BOOL" iec_addr="%QX288.10" expanded="false" mb_access="ro" explicitAccess="false"/>
				<pfc_var name="FRM_PORT_LAMP_TEST_PB_cfg" comment="" data_type="BOOL" iec_addr="%QX288.11" expanded="false" mb_access="ro" explicitAccess="false"/>
				<pfc_var name="FRM_STBD_LAMP_TEST_PB_cfg" comment="" data_type="BOOL" iec_addr="%QX288.12" expanded="false" mb_access="ro" explicitAccess="false"/>
				<pfc_var name="FRM_ENG_TURNING_AHEAD_cfg" comment="" data_type="BOOL" iec_addr="%QX288.3" expanded="false" mb_access="ro" explicitAccess="false"/>
				<pfc_var name="FRM_ENG_TURNING_AST_cfg" comment="" data_type="BOOL" iec_addr="%QX288.4" expanded="false" mb_access="ro" explicitAccess="false"/>
				<pfc_var name="FRM_ENG_SENSOR_1_FAILURE_cfg" comment="" data_type="BOOL" iec_addr="%QX286.8" expanded="false" mb_access="ro" explicitAccess="false"/>
				<pfc_var name="FRM_ECR_MAN_CONTROL_cfg" comment="" data_type="BOOL" iec_addr="%QX285.2" expanded="false" mb_access="ro" explicitAccess="false"/>
				<pfc_var name="FRM_LOCAL_MAN_CONTROL_cfg" comment="" data_type="BOOL" iec_addr="%QX285.3" expanded="false" mb_access="ro" explicitAccess="false"/>
				<pfc_var name="FRM_FAIL_ACOUSTIC_cfg" comment="" data_type="BOOL" iec_addr="%QX289.13" expanded="false" mb_access="ro" explicitAccess="false"/>
				<pfc_var name="FRM_CONTROL_TRANS_BUZZER_BRG_cfg" comment="" data_type="BOOL" iec_addr="%QX389.14" expanded="false" mb_access="ro" explicitAccess="false"/>
				<pfc_var name="FRM_CONTROL_TRANS_BUZZER_MCR_cfg" comment="" data_type="BOOL" iec_addr="%QX389.15" expanded="false" mb_access="ro" explicitAccess="false"/>
			</pfc_vars>
			<k_bus comment="" expanded="false">
				<terminal article-no="0750-0636" comment="" expanded="false" is_array_mode="false">
					<variable name="xVar_0_0" comment="moving negative" expanded="false" mb_access="unused" explicitAccess="false"/>
					<variable name="xVar_0_1" comment="moving positive" expanded="false" mb_access="unused" explicitAccess="false"/>
					<variable name="xVar_0_2" comment="On target" expanded="false" mb_access="unused" explicitAccess="false"/>
					<variable name="xVar_0_3" comment="busy" expanded="false" mb_access="unused" explicitAccess="false"/>
					<variable name="xVar_0_4" comment="standstill" expanded="false" mb_access="unused" explicitAccess="false"/>
					<variable name="xVar_0_5" comment="reference ok" expanded="false" mb_access="unused" explicitAccess="false"/>
					<variable name="xVar_0_6" comment="error, see extended info" expanded="false" mb_access="unused" explicitAccess="false"/>
					<variable name="xVar_0_7" comment="preset input enabled" expanded="false" mb_access="unused" explicitAccess="false"/>
					<variable name="xVar_0_8" comment="optimize on (and Z-Input for 750-636 &gt; FW2)" expanded="false" mb_access="unused" explicitAccess="false"/>
					<variable name="xVar_0_9" comment="extended info on" expanded="false" mb_access="unused" explicitAccess="false"/>
					<variable name="xVar_0_10" comment="PWM active" expanded="false" mb_access="unused" explicitAccess="false"/>
					<variable name="xVar_0_11" comment="current control on" expanded="false" mb_access="unused" explicitAccess="false"/>
					<variable name="xVar_0_12" comment="preset input" expanded="false" mb_access="unused" explicitAccess="false"/>
					<variable name="xVar_0_13" comment="limit switch negative" expanded="false" mb_access="unused" explicitAccess="false"/>
					<variable name="xVar_0_14" comment="limit switch positive" expanded="false" mb_access="unused" explicitAccess="false"/>
					<variable name="wVar_0_15" comment="actual position low word" expanded="false" mb_access="unused" explicitAccess="false"/>
					<variable name="xVar_0_16" comment="over temperature warning" expanded="false" mb_access="unused" explicitAccess="false"/>
					<variable name="xVar_0_17" comment="over temperature" expanded="false" mb_access="unused" explicitAccess="false"/>
					<variable name="xVar_0_18" comment="overflow warning" expanded="false" mb_access="unused" explicitAccess="false"/>
					<variable name="xVar_0_19" comment="24V ok" expanded="false" mb_access="unused" explicitAccess="false"/>
					<variable name="xVar_0_20" comment="overload" expanded="false" mb_access="unused" explicitAccess="false"/>
					<variable name="xVar_0_21" comment="motion detection timeout" expanded="false" mb_access="unused" explicitAccess="false"/>
					<variable name="xVar_0_22" comment="parameter write failed" expanded="false" mb_access="unused" explicitAccess="false"/>
					<variable name="xVar_0_23" comment="24VL Ok (only 750-636/000-800)" expanded="false" mb_access="unused" explicitAccess="false"/>
					<variable name="xVar_0_24" comment="24VM Ok  (only 750-636/000-800)" expanded="false" mb_access="unused" explicitAccess="false"/>
					<variable name="wVar_0_25" comment="actual position high word" expanded="false" mb_access="unused" explicitAccess="false"/>
					<variable name="xVar_0_26" comment="move negative" expanded="false" mb_access="unused" explicitAccess="false"/>
					<variable name="xVar_0_27" comment="move positive" expanded="false" mb_access="unused" explicitAccess="false"/>
					<variable name="xVar_0_28" comment="positioning" expanded="false" mb_access="unused" explicitAccess="false"/>
					<variable name="xVar_0_29" comment="preset" expanded="false" mb_access="unused" explicitAccess="false"/>
					<variable name="xVar_0_30" comment="current control on" expanded="false" mb_access="unused" explicitAccess="false"/>
					<variable name="xVar_0_31" comment="preset input enable" expanded="false" mb_access="unused" explicitAccess="false"/>
					<variable name="xVar_0_32" comment="optimize on" expanded="false" mb_access="unused" explicitAccess="false"/>
					<variable name="xVar_0_33" comment="extended info on" expanded="false" mb_access="unused" explicitAccess="false"/>
					<variable name="xVar_0_34" comment="error quit" expanded="false" mb_access="unused" explicitAccess="false"/>
					<variable name="wVar_0_35" comment="target position low word" expanded="false" mb_access="unused" explicitAccess="false"/>
					<variable name="wVar_0_36" comment="target position high word" expanded="false" mb_access="unused" explicitAccess="false"/>
				</terminal>
				<terminal article-no="0750-9999/0400-0008" comment="" expanded="false" is_array_mode="false">
					<variable name="xVar_1_0" comment="Ch_1 Digital input" expanded="false" mb_access="unused" explicitAccess="false"/>
					<variable name="xVar_1_1" comment="Ch_2 Digital input" expanded="false" mb_access="unused" explicitAccess="false"/>
					<variable name="xVar_1_2" comment="Ch_3 Digital input" expanded="false" mb_access="unused" explicitAccess="false"/>
					<variable name="xVar_1_3" comment="Ch_4 Digital input" expanded="false" mb_access="unused" explicitAccess="false"/>
					<variable name="xVar_1_4" comment="Ch_5 Digital input" expanded="false" mb_access="unused" explicitAccess="false"/>
					<variable name="xVar_1_5" comment="Ch_6 Digital input" expanded="false" mb_access="unused" explicitAccess="false"/>
					<variable name="xVar_1_6" comment="Ch_7 Digital input" expanded="false" mb_access="unused" explicitAccess="false"/>
					<variable name="xVar_1_7" comment="Ch_8 Digital input" expanded="false" mb_access="unused" explicitAccess="false"/>
				</terminal>
				<terminal article-no="0750-9999/0400-0008" comment="" expanded="false" is_array_mode="false">
					<variable name="xVar_2_0" comment="Ch_1 Digital input" expanded="false" mb_access="unused" explicitAccess="false"/>
					<variable name="xVar_2_1" comment="Ch_2 Digital input" expanded="false" mb_access="unused" explicitAccess="false"/>
					<variable name="xVar_2_2" comment="Ch_3 Digital input" expanded="false" mb_access="unused" explicitAccess="false"/>
					<variable name="xVar_2_3" comment="Ch_4 Digital input" expanded="false" mb_access="unused" explicitAccess="false"/>
					<variable name="xVar_2_4" comment="Ch_5 Digital input" expanded="false" mb_access="unused" explicitAccess="false"/>
					<variable name="xVar_2_5" comment="Ch_6 Digital input" expanded="false" mb_access="unused" explicitAccess="false"/>
					<variable name="xVar_2_6" comment="Ch_7 Digital input" expanded="false" mb_access="unused" explicitAccess="false"/>
					<variable name="xVar_2_7" comment="Ch_8 Digital input" expanded="false" mb_access="unused" explicitAccess="false"/>
				</terminal>
				<terminal article-no="0750-9999/0400-0008" comment="" expanded="false" is_array_mode="false">
					<variable name="xVar_3_0" comment="Ch_1 Digital input" expanded="false" mb_access="unused" explicitAccess="false"/>
					<variable name="xVar_3_1" comment="Ch_2 Digital input" expanded="false" mb_access="unused" explicitAccess="false"/>
					<variable name="xVar_3_2" comment="Ch_3 Digital input" expanded="false" mb_access="unused" explicitAccess="false"/>
					<variable name="xVar_3_3" comment="Ch_4 Digital input" expanded="false" mb_access="unused" explicitAccess="false"/>
					<variable name="xVar_3_4" comment="Ch_5 Digital input" expanded="false" mb_access="unused" explicitAccess="false"/>
					<variable name="xVar_3_5" comment="Ch_6 Digital input" expanded="false" mb_access="unused" explicitAccess="false"/>
					<variable name="xVar_3_6" comment="Ch_7 Digital input" expanded="false" mb_access="unused" explicitAccess="false"/>
					<variable name="xVar_3_7" comment="Ch_8 Digital input" expanded="false" mb_access="unused" explicitAccess="false"/>
				</terminal>
				<terminal article-no="0750-9999/0400-0008" comment="" expanded="false" is_array_mode="false">
					<variable name="xVar_4_0" comment="Ch_1 Digital input" expanded="false" mb_access="unused" explicitAccess="false"/>
					<variable name="xVar_4_1" comment="Ch_2 Digital input" expanded="false" mb_access="unused" explicitAccess="false"/>
					<variable name="xVar_4_2" comment="Ch_3 Digital input" expanded="false" mb_access="unused" explicitAccess="false"/>
					<variable name="xVar_4_3" comment="Ch_4 Digital input" expanded="false" mb_access="unused" explicitAccess="false"/>
					<variable name="xVar_4_4" comment="Ch_5 Digital input" expanded="false" mb_access="unused" explicitAccess="false"/>
					<variable name="xVar_4_5" comment="Ch_6 Digital input" expanded="false" mb_access="unused" explicitAccess="false"/>
					<variable name="xVar_4_6" comment="Ch_7 Digital input" expanded="false" mb_access="unused" explicitAccess="false"/>
					<variable name="xVar_4_7" comment="Ch_8 Digital input" expanded="false" mb_access="unused" explicitAccess="false"/>
				</terminal>
				<terminal article-no="0750-9999/0500-0008" comment="" expanded="false" is_array_mode="false">
					<variable name="xVar_5_0" comment="Ch_1 Digital output" expanded="false" mb_access="unused" explicitAccess="false"/>
					<variable name="xVar_5_1" comment="Ch_2 Digital output" expanded="false" mb_access="unused" explicitAccess="false"/>
					<variable name="xVar_5_2" comment="Ch_3 Digital output" expanded="false" mb_access="unused" explicitAccess="false"/>
					<variable name="xVar_5_3" comment="Ch_4 Digital output" expanded="false" mb_access="unused" explicitAccess="false"/>
					<variable name="xVar_5_4" comment="Ch_5 Digital output" expanded="false" mb_access="unused" explicitAccess="false"/>
					<variable name="xVar_5_5" comment="Ch_6 Digital output" expanded="false" mb_access="unused" explicitAccess="false"/>
					<variable name="xVar_5_6" comment="Ch_7 Digital output" expanded="false" mb_access="unused" explicitAccess="false"/>
					<variable name="xVar_5_7" comment="Ch_8 Digital output" expanded="false" mb_access="unused" explicitAccess="false"/>
				</terminal>
				<terminal article-no="0750-9999/0500-0008" comment="" expanded="false" is_array_mode="false">
					<variable name="xVar_6_0" comment="Ch_1 Digital output" expanded="false" mb_access="unused" explicitAccess="false"/>
					<variable name="xVar_6_1" comment="Ch_2 Digital output" expanded="false" mb_access="unused" explicitAccess="false"/>
					<variable name="xVar_6_2" comment="Ch_3 Digital output" expanded="false" mb_access="unused" explicitAccess="false"/>
					<variable name="xVar_6_3" comment="Ch_4 Digital output" expanded="false" mb_access="unused" explicitAccess="false"/>
					<variable name="xVar_6_4" comment="Ch_5 Digital output" expanded="false" mb_access="unused" explicitAccess="false"/>
					<variable name="xVar_6_5" comment="Ch_6 Digital output" expanded="false" mb_access="unused" explicitAccess="false"/>
					<variable name="xVar_6_6" comment="Ch_7 Digital output" expanded="false" mb_access="unused" explicitAccess="false"/>
					<variable name="xVar_6_7" comment="Ch_8 Digital output" expanded="false" mb_access="unused" explicitAccess="false"/>
				</terminal>
				<terminal article-no="0750-9999/0500-0008" comment="" expanded="false" is_array_mode="false">
					<variable name="xVar_7_0" comment="Ch_1 Digital output" expanded="false" mb_access="unused" explicitAccess="false"/>
					<variable name="xVar_7_1" comment="Ch_2 Digital output" expanded="false" mb_access="unused" explicitAccess="false"/>
					<variable name="xVar_7_2" comment="Ch_3 Digital output" expanded="false" mb_access="unused" explicitAccess="false"/>
					<variable name="xVar_7_3" comment="Ch_4 Digital output" expanded="false" mb_access="unused" explicitAccess="false"/>
					<variable name="xVar_7_4" comment="Ch_5 Digital output" expanded="false" mb_access="unused" explicitAccess="false"/>
					<variable name="xVar_7_5" comment="Ch_6 Digital output" expanded="false" mb_access="unused" explicitAccess="false"/>
					<variable name="xVar_7_6" comment="Ch_7 Digital output" expanded="false" mb_access="unused" explicitAccess="false"/>
					<variable name="xVar_7_7" comment="Ch_8 Digital output" expanded="false" mb_access="unused" explicitAccess="false"/>
				</terminal>
				<terminal article-no="0750-9999/0500-0008" comment="" expanded="false" is_array_mode="false">
					<variable name="xVar_8_0" comment="Ch_1 Digital output" expanded="false" mb_access="unused" explicitAccess="false"/>
					<variable name="xVar_8_1" comment="Ch_2 Digital output" expanded="false" mb_access="unused" explicitAccess="false"/>
					<variable name="xVar_8_2" comment="Ch_3 Digital output" expanded="false" mb_access="unused" explicitAccess="false"/>
					<variable name="xVar_8_3" comment="Ch_4 Digital output" expanded="false" mb_access="unused" explicitAccess="false"/>
					<variable name="xVar_8_4" comment="Ch_5 Digital output" expanded="false" mb_access="unused" explicitAccess="false"/>
					<variable name="xVar_8_5" comment="Ch_6 Digital output" expanded="false" mb_access="unused" explicitAccess="false"/>
					<variable name="xVar_8_6" comment="Ch_7 Digital output" expanded="false" mb_access="unused" explicitAccess="false"/>
					<variable name="xVar_8_7" comment="Ch_8 Digital output" expanded="false" mb_access="unused" explicitAccess="false"/>
				</terminal>
				<terminal article-no="0750-9999/0500-0008" comment="" expanded="false" is_array_mode="false">
					<variable name="xVar_9_0" comment="Ch_1 Digital output" expanded="false" mb_access="unused" explicitAccess="false"/>
					<variable name="xVar_9_1" comment="Ch_2 Digital output" expanded="false" mb_access="unused" explicitAccess="false"/>
					<variable name="xVar_9_2" comment="Ch_3 Digital output" expanded="false" mb_access="unused" explicitAccess="false"/>
					<variable name="xVar_9_3" comment="Ch_4 Digital output" expanded="false" mb_access="unused" explicitAccess="false"/>
					<variable name="xVar_9_4" comment="Ch_5 Digital output" expanded="false" mb_access="unused" explicitAccess="false"/>
					<variable name="xVar_9_5" comment="Ch_6 Digital output" expanded="false" mb_access="unused" explicitAccess="false"/>
					<variable name="xVar_9_6" comment="Ch_7 Digital output" expanded="false" mb_access="unused" explicitAccess="false"/>
					<variable name="xVar_9_7" comment="Ch_8 Digital output" expanded="false" mb_access="unused" explicitAccess="false"/>
				</terminal>
				<terminal article-no="0753-0555" comment="" expanded="false" is_array_mode="false">
					<variable name="wVar_10_0" comment="Ch_1 Analog output" expanded="false" mb_access="unused" explicitAccess="false"/>
					<variable name="wVar_10_1" comment="Ch_2 Analog output" expanded="false" mb_access="unused" explicitAccess="false"/>
					<variable name="wVar_10_2" comment="Ch_3 Analog output" expanded="false" mb_access="unused" explicitAccess="false"/>
					<variable name="wVar_10_3" comment="Ch_4 Analog output" expanded="false" mb_access="unused" explicitAccess="false"/>
				</terminal>
				<terminal article-no="0753-0555" comment="" expanded="false" is_array_mode="false">
					<variable name="wVar_11_0" comment="Ch_1 Analog output" expanded="false" mb_access="unused" explicitAccess="false"/>
					<variable name="wVar_11_1" comment="Ch_2 Analog output" expanded="false" mb_access="unused" explicitAccess="false"/>
					<variable name="wVar_11_2" comment="Ch_3 Analog output" expanded="false" mb_access="unused" explicitAccess="false"/>
					<variable name="wVar_11_3" comment="Ch_4 Analog output" expanded="false" mb_access="unused" explicitAccess="false"/>
				</terminal>
				<terminal article-no="0753-0555" comment="" expanded="false" is_array_mode="false">
					<variable name="wVar_12_0" comment="Ch_1 Analog output" expanded="false" mb_access="unused" explicitAccess="false"/>
					<variable name="wVar_12_1" comment="Ch_2 Analog output" expanded="false" mb_access="unused" explicitAccess="false"/>
					<variable name="wVar_12_2" comment="Ch_3 Analog output" expanded="false" mb_access="unused" explicitAccess="false"/>
					<variable name="wVar_12_3" comment="Ch_4 Analog output" expanded="false" mb_access="unused" explicitAccess="false"/>
				</terminal>
				<terminal article-no="0753-0555" comment="" expanded="false" is_array_mode="false">
					<variable name="wVar_13_0" comment="Ch_1 Analog output" expanded="false" mb_access="unused" explicitAccess="false"/>
					<variable name="wVar_13_1" comment="Ch_2 Analog output" expanded="false" mb_access="unused" explicitAccess="false"/>
					<variable name="wVar_13_2" comment="Ch_3 Analog output" expanded="false" mb_access="unused" explicitAccess="false"/>
					<variable name="wVar_13_3" comment="Ch_4 Analog output" expanded="false" mb_access="unused" explicitAccess="false"/>
				</terminal>
				<terminal article-no="0750-0452" comment="" expanded="false" is_array_mode="false">
					<variable name="wVar_14_0" comment="Ch_1 Input word" expanded="false" mb_access="unused" explicitAccess="false"/>
					<variable name="wVar_14_1" comment="Ch_2 Input word" expanded="false" mb_access="unused" explicitAccess="false"/>
				</terminal>
				<terminal article-no="0750-0452" comment="" expanded="false" is_array_mode="false">
					<variable name="wVar_15_0" comment="Ch_1 Input word" expanded="false" mb_access="unused" explicitAccess="false"/>
					<variable name="wVar_15_1" comment="Ch_2 Input word" expanded="false" mb_access="unused" explicitAccess="false"/>
				</terminal>
			</k_bus>
		</mb_slave>
		<mb_slave comment="Ethernet MR Controller 100MBit 2Port" name="ESS" expanded="true" type="wago" article-no="0750-0882">
			<mb_connection type="eth" transport="TCP" port="502" ip="192.168.1.2" unitid="2" request_delay_ms="0" response_timeout_ms="20"/>
			<service_connection type="eth" ip="192.168.1.2"/>
			<generic_vars comment="" expanded="false"/>
			<pfc_vars comment="" expanded="true">
				<pfc_var name="ESS_BR_ALARM_ACK_cfg" comment="" data_type="BOOL" iec_addr="%QX274.1" expanded="false" mb_access="ro" explicitAccess="false"/>
				<pfc_var name="ESS_ECR_ALARM_ACK_cfg" comment="" data_type="BOOL" iec_addr="%QX274.2" expanded="false" mb_access="ro" explicitAccess="false"/>
				<pfc_var name="ESS_PORT_ALARM_ACK_cfg" comment="" data_type="BOOL" iec_addr="%QX274.3" expanded="false" mb_access="ro" explicitAccess="false"/>
				<pfc_var name="ESS_STBD_ALARM_ACK_cfg" comment="" data_type="BOOL" iec_addr="%QX274.4" expanded="false" mb_access="ro" explicitAccess="false"/>
				<pfc_var name="ESS_ENG_TURNING_AHEAD_cfg" comment="" data_type="BOOL" iec_addr="%QX272.0" expanded="false" mb_access="ro" explicitAccess="false"/>
				<pfc_var name="ESS_ENG_TURNING_AST_cfg" comment="" data_type="BOOL" iec_addr="%QX272.1" expanded="false" mb_access="ro" explicitAccess="false"/>
				<pfc_var name="ESS_ENG_SENSOR_1_FAILURE_cfg" comment="" data_type="BOOL" iec_addr="%QX272.3" expanded="false" mb_access="ro" explicitAccess="false"/>
			</pfc_vars>
			<k_bus comment="" expanded="false"/>
		</mb_slave>
	</master_interface>
</network>
                              
*)                                 
;                                  
END_PROGRAM

(* POU Generated Code/Ethernet/MBCFG_RCS, ST *)
PROGRAM MBCFG_RCS(* generated by config one prg for each slave *)

VAR_INPUT

END_VAR

VAR_OUTPUT
       FRM_BR_CONTROL_cfg       :    BOOL;       (**) 
       FRM_ECR_AUT_CONTROL_cfg       :    BOOL;       (**) 
       FRM_ECR_LAMP_TEST_PB_cfg       :    BOOL;       (**) 
       FRM_BR_LAMP_TEST_PB_cfg       :    BOOL;       (**) 
       FRM_PORT_LAMP_TEST_PB_cfg       :    BOOL;       (**) 
       FRM_STBD_LAMP_TEST_PB_cfg       :    BOOL;       (**) 
       FRM_ENG_TURNING_AHEAD_cfg       :    BOOL;       (**) 
       FRM_ENG_TURNING_AST_cfg       :    BOOL;       (**) 
       FRM_ENG_SENSOR_1_FAILURE_cfg       :    BOOL;       (**) 
       FRM_ECR_MAN_CONTROL_cfg       :    BOOL;       (**) 
       FRM_LOCAL_MAN_CONTROL_cfg       :    BOOL;       (**) 
       FRM_FAIL_ACOUSTIC_cfg       :    BOOL;       (**) 
       FRM_CONTROL_TRANS_BUZZER_BRG_cfg       :    BOOL;       (**) 
       FRM_CONTROL_TRANS_BUZZER_MCR_cfg       :    BOOL;       (**) 

    (*--- system variables (read only) ----------------------------------------*)
    MBCFG_IpAddress     :   STRING(11) := '192.168.1.1'; (* address of this slave *)
    MBCFG_Port          :   UINT := 502;               (* IP - Port *)
    MBCFG_UnitID        :   BYTE := 1;             (* MODBUS Unit-Id *)
    MBCFG_TimeOut       :   TIME := t#20ms;           (* Response timeout*)
	MBCFG_RequestDelay  :   TIME  := t#0ms;         (* 0 means no delay *)
    MBCFG_Error         :   MBCFG_eERROR := MBCFG_START_UP;
	MBCFG_LastJob       :   MBCFG_typCOM_JOB;
    (*-------------------------------------------------------------------------*)
END_VAR

{library private}
VAR CONSTANT
    zz_VARIABLECOUNT:   INT := 14; (* number of variables  *)
    zz_JOBCOUNT     :   INT := 2; (* number of jobs *)
END_VAR
VAR

    (*=== VARIABLE LIST ===============================================================================*)
    zz_VariableList :   ARRAY[1..zz_VARIABLECOUNT] OF MBCFG_typVARIABLE :=
    (    DataType        := MBCFG_TYPE_BOOL,
        ByteOrder       := MBCFG_BYTE_ORDER_0,
        BitSize         := 1,
        ptVar           := 0,
        ReadJobIndex    := 1,
        ReadStartBitNo  := 0,
        WriteJobIndex   := 0,
        WriteStartBitNo := 0 ),
    (    DataType        := MBCFG_TYPE_BOOL,
        ByteOrder       := MBCFG_BYTE_ORDER_0,
        BitSize         := 1,
        ptVar           := 0,
        ReadJobIndex    := 1,
        ReadStartBitNo  := 1,
        WriteJobIndex   := 0,
        WriteStartBitNo := 0 ),
    (    DataType        := MBCFG_TYPE_BOOL,
        ByteOrder       := MBCFG_BYTE_ORDER_0,
        BitSize         := 1,
        ptVar           := 0,
        ReadJobIndex    := 1,
        ReadStartBitNo  := 57,
        WriteJobIndex   := 0,
        WriteStartBitNo := 0 ),
    (    DataType        := MBCFG_TYPE_BOOL,
        ByteOrder       := MBCFG_BYTE_ORDER_0,
        BitSize         := 1,
        ptVar           := 0,
        ReadJobIndex    := 1,
        ReadStartBitNo  := 58,
        WriteJobIndex   := 0,
        WriteStartBitNo := 0 ),
    (    DataType        := MBCFG_TYPE_BOOL,
        ByteOrder       := MBCFG_BYTE_ORDER_0,
        BitSize         := 1,
        ptVar           := 0,
        ReadJobIndex    := 1,
        ReadStartBitNo  := 59,
        WriteJobIndex   := 0,
        WriteStartBitNo := 0 ),
    (    DataType        := MBCFG_TYPE_BOOL,
        ByteOrder       := MBCFG_BYTE_ORDER_0,
        BitSize         := 1,
        ptVar           := 0,
        ReadJobIndex    := 1,
        ReadStartBitNo  := 60,
        WriteJobIndex   := 0,
        WriteStartBitNo := 0 ),
    (    DataType        := MBCFG_TYPE_BOOL,
        ByteOrder       := MBCFG_BYTE_ORDER_0,
        BitSize         := 1,
        ptVar           := 0,
        ReadJobIndex    := 1,
        ReadStartBitNo  := 51,
        WriteJobIndex   := 0,
        WriteStartBitNo := 0 ),
    (    DataType        := MBCFG_TYPE_BOOL,
        ByteOrder       := MBCFG_BYTE_ORDER_0,
        BitSize         := 1,
        ptVar           := 0,
        ReadJobIndex    := 1,
        ReadStartBitNo  := 52,
        WriteJobIndex   := 0,
        WriteStartBitNo := 0 ),
    (    DataType        := MBCFG_TYPE_BOOL,
        ByteOrder       := MBCFG_BYTE_ORDER_0,
        BitSize         := 1,
        ptVar           := 0,
        ReadJobIndex    := 1,
        ReadStartBitNo  := 24,
        WriteJobIndex   := 0,
        WriteStartBitNo := 0 ),
    (    DataType        := MBCFG_TYPE_BOOL,
        ByteOrder       := MBCFG_BYTE_ORDER_0,
        BitSize         := 1,
        ptVar           := 0,
        ReadJobIndex    := 1,
        ReadStartBitNo  := 2,
        WriteJobIndex   := 0,
        WriteStartBitNo := 0 ),
    (    DataType        := MBCFG_TYPE_BOOL,
        ByteOrder       := MBCFG_BYTE_ORDER_0,
        BitSize         := 1,
        ptVar           := 0,
        ReadJobIndex    := 1,
        ReadStartBitNo  := 3,
        WriteJobIndex   := 0,
        WriteStartBitNo := 0 ),
    (    DataType        := MBCFG_TYPE_BOOL,
        ByteOrder       := MBCFG_BYTE_ORDER_0,
        BitSize         := 1,
        ptVar           := 0,
        ReadJobIndex    := 1,
        ReadStartBitNo  := 77,
        WriteJobIndex   := 0,
        WriteStartBitNo := 0 ),
    (    DataType        := MBCFG_TYPE_BOOL,
        ByteOrder       := MBCFG_BYTE_ORDER_0,
        BitSize         := 1,
        ptVar           := 0,
        ReadJobIndex    := 2,
        ReadStartBitNo  := 0,
        WriteJobIndex   := 0,
        WriteStartBitNo := 0 ),
    (    DataType        := MBCFG_TYPE_BOOL,
        ByteOrder       := MBCFG_BYTE_ORDER_0,
        BitSize         := 1,
        ptVar           := 0,
        ReadJobIndex    := 2,
        ReadStartBitNo  := 1,
        WriteJobIndex   := 0,
        WriteStartBitNo := 0 )

                        ;
    (*=================================================================================================*)

    (*=== JOB LIST ====================================================================================*)
    zz_JobList     :   ARRAY[1..zz_JOBCOUNT] OF MBCFG_typCOM_JOB :=
     (   Functioncode            := 2,
        ReadStartAddress        := 4560,
        ReadQuantity            := 78,
        WriteStartAddress       := 0,
        WriteQuantity           := 0,
        ptReadData              := 0, 
        ptWriteData             := 0 ),
     (   Functioncode            := 2,
        ReadStartAddress        := 6238,
        ReadQuantity            := 2,
        WriteStartAddress       := 0,
        WriteQuantity           := 0,
        ptReadData              := 0, 
        ptWriteData             := 0 )

                        ;
    (*=================================================================================================*)

    (*=== DATA FIELDS =================================================================================*)
     zz_DataField_1_Read       :       ARRAY[1..5] OF WORD;
     zz_DataField_2_Read       :       ARRAY[1..1] OF WORD;
	
    (*=================================================================================================*)

    (*=== MODBUS MASTER =====================================*)
    zz_MBCFG_MASTER_ETH :       MBCFG_MASTER_TCP;
    (*=======================================================*)

END_VAR
(*--- for each variable -------------------------*)
   zz_VariableList[1].ptVar := ADR(FRM_BR_CONTROL_cfg);
   zz_VariableList[2].ptVar := ADR(FRM_ECR_AUT_CONTROL_cfg);
   zz_VariableList[3].ptVar := ADR(FRM_ECR_LAMP_TEST_PB_cfg);
   zz_VariableList[4].ptVar := ADR(FRM_BR_LAMP_TEST_PB_cfg);
   zz_VariableList[5].ptVar := ADR(FRM_PORT_LAMP_TEST_PB_cfg);
   zz_VariableList[6].ptVar := ADR(FRM_STBD_LAMP_TEST_PB_cfg);
   zz_VariableList[7].ptVar := ADR(FRM_ENG_TURNING_AHEAD_cfg);
   zz_VariableList[8].ptVar := ADR(FRM_ENG_TURNING_AST_cfg);
   zz_VariableList[9].ptVar := ADR(FRM_ENG_SENSOR_1_FAILURE_cfg);
   zz_VariableList[10].ptVar := ADR(FRM_ECR_MAN_CONTROL_cfg);
   zz_VariableList[11].ptVar := ADR(FRM_LOCAL_MAN_CONTROL_cfg);
   zz_VariableList[12].ptVar := ADR(FRM_FAIL_ACOUSTIC_cfg);
   zz_VariableList[13].ptVar := ADR(FRM_CONTROL_TRANS_BUZZER_BRG_cfg);
   zz_VariableList[14].ptVar := ADR(FRM_CONTROL_TRANS_BUZZER_MCR_cfg);

(*-----------------------------------------------*)

(*--- for each job -----------------------------------*)
zz_JobList[1].ptReadData   := ADR(zz_DataField_1_Read);
zz_JobList[2].ptReadData   := ADR(zz_DataField_2_Read);

(*----------------------------------------------------*)


(*#### START OF FIXED CODE #####################################*)
zz_MBCFG_MASTER_ETH(	strIpAddress    := MBCFG_IpAddress,                 (* fixed entry     *)
                        uiPort          := MBCFG_Port,                      (* fixed entry     *)
                        bUnitID         := MBCFG_UnitID,                    (* fixed entry     *)
                        tTimeOut        := MBCFG_TimeOut,                   (* fixed entry     *)
                        iVariableCount  := zz_VARIABLECOUNT,
                        ptVariableList  := ADR(zz_VariableList),
                        iJobCount       := zz_JOBCOUNT,
                        ptJobList       := ADR(zz_JobList),
                        tRequestDelay   := MBCFG_RequestDelay,              (* fixed entry     *)
                        eError          => MBCFG_Error,                     (* fixed entry     *)
                        LastJob         => MBCFG_LastJob                    (* fixed entry     *)
                    );
(*##############################################################*)
END_PROGRAM

(* POU Generated Code/Ethernet/MBCFG_ESS, ST *)
PROGRAM MBCFG_ESS(* generated by config one prg for each slave *)

VAR_INPUT

END_VAR

VAR_OUTPUT
       ESS_BR_ALARM_ACK_cfg       :    BOOL;       (**) 
       ESS_ECR_ALARM_ACK_cfg       :    BOOL;       (**) 
       ESS_PORT_ALARM_ACK_cfg       :    BOOL;       (**) 
       ESS_STBD_ALARM_ACK_cfg       :    BOOL;       (**) 
       ESS_ENG_TURNING_AHEAD_cfg       :    BOOL;       (**) 
       ESS_ENG_TURNING_AST_cfg       :    BOOL;       (**) 
       ESS_ENG_SENSOR_1_FAILURE_cfg       :    BOOL;       (**) 

    (*--- system variables (read only) ----------------------------------------*)
    MBCFG_IpAddress     :   STRING(11) := '192.168.1.2'; (* address of this slave *)
    MBCFG_Port          :   UINT := 502;               (* IP - Port *)
    MBCFG_UnitID        :   BYTE := 2;             (* MODBUS Unit-Id *)
    MBCFG_TimeOut       :   TIME := t#20ms;           (* Response timeout*)
	MBCFG_RequestDelay  :   TIME  := t#0ms;         (* 0 means no delay *)
    MBCFG_Error         :   MBCFG_eERROR := MBCFG_START_UP;
	MBCFG_LastJob       :   MBCFG_typCOM_JOB;
    (*-------------------------------------------------------------------------*)
END_VAR

{library private}
VAR CONSTANT
    zz_VARIABLECOUNT:   INT := 7; (* number of variables  *)
    zz_JOBCOUNT     :   INT := 1; (* number of jobs *)
END_VAR
VAR

    (*=== VARIABLE LIST ===============================================================================*)
    zz_VariableList :   ARRAY[1..zz_VARIABLECOUNT] OF MBCFG_typVARIABLE :=
    (    DataType        := MBCFG_TYPE_BOOL,
        ByteOrder       := MBCFG_BYTE_ORDER_0,
        BitSize         := 1,
        ptVar           := 0,
        ReadJobIndex    := 1,
        ReadStartBitNo  := 33,
        WriteJobIndex   := 0,
        WriteStartBitNo := 0 ),
    (    DataType        := MBCFG_TYPE_BOOL,
        ByteOrder       := MBCFG_BYTE_ORDER_0,
        BitSize         := 1,
        ptVar           := 0,
        ReadJobIndex    := 1,
        ReadStartBitNo  := 34,
        WriteJobIndex   := 0,
        WriteStartBitNo := 0 ),
    (    DataType        := MBCFG_TYPE_BOOL,
        ByteOrder       := MBCFG_BYTE_ORDER_0,
        BitSize         := 1,
        ptVar           := 0,
        ReadJobIndex    := 1,
        ReadStartBitNo  := 35,
        WriteJobIndex   := 0,
        WriteStartBitNo := 0 ),
    (    DataType        := MBCFG_TYPE_BOOL,
        ByteOrder       := MBCFG_BYTE_ORDER_0,
        BitSize         := 1,
        ptVar           := 0,
        ReadJobIndex    := 1,
        ReadStartBitNo  := 36,
        WriteJobIndex   := 0,
        WriteStartBitNo := 0 ),
    (    DataType        := MBCFG_TYPE_BOOL,
        ByteOrder       := MBCFG_BYTE_ORDER_0,
        BitSize         := 1,
        ptVar           := 0,
        ReadJobIndex    := 1,
        ReadStartBitNo  := 0,
        WriteJobIndex   := 0,
        WriteStartBitNo := 0 ),
    (    DataType        := MBCFG_TYPE_BOOL,
        ByteOrder       := MBCFG_BYTE_ORDER_0,
        BitSize         := 1,
        ptVar           := 0,
        ReadJobIndex    := 1,
        ReadStartBitNo  := 1,
        WriteJobIndex   := 0,
        WriteStartBitNo := 0 ),
    (    DataType        := MBCFG_TYPE_BOOL,
        ByteOrder       := MBCFG_BYTE_ORDER_0,
        BitSize         := 1,
        ptVar           := 0,
        ReadJobIndex    := 1,
        ReadStartBitNo  := 3,
        WriteJobIndex   := 0,
        WriteStartBitNo := 0 )

                        ;
    (*=================================================================================================*)

    (*=== JOB LIST ====================================================================================*)
    zz_JobList     :   ARRAY[1..zz_JOBCOUNT] OF MBCFG_typCOM_JOB :=
     (   Functioncode            := 2,
        ReadStartAddress        := 4352,
        ReadQuantity            := 37,
        WriteStartAddress       := 0,
        WriteQuantity           := 0,
        ptReadData              := 0, 
        ptWriteData             := 0 )

                        ;
    (*=================================================================================================*)

    (*=== DATA FIELDS =================================================================================*)
     zz_DataField_1_Read       :       ARRAY[1..3] OF WORD;
	
    (*=================================================================================================*)

    (*=== MODBUS MASTER =====================================*)
    zz_MBCFG_MASTER_ETH :       MBCFG_MASTER_TCP;
    (*=======================================================*)

END_VAR
(*--- for each variable -------------------------*)
   zz_VariableList[1].ptVar := ADR(ESS_BR_ALARM_ACK_cfg);
   zz_VariableList[2].ptVar := ADR(ESS_ECR_ALARM_ACK_cfg);
   zz_VariableList[3].ptVar := ADR(ESS_PORT_ALARM_ACK_cfg);
   zz_VariableList[4].ptVar := ADR(ESS_STBD_ALARM_ACK_cfg);
   zz_VariableList[5].ptVar := ADR(ESS_ENG_TURNING_AHEAD_cfg);
   zz_VariableList[6].ptVar := ADR(ESS_ENG_TURNING_AST_cfg);
   zz_VariableList[7].ptVar := ADR(ESS_ENG_SENSOR_1_FAILURE_cfg);

(*-----------------------------------------------*)

(*--- for each job -----------------------------------*)
zz_JobList[1].ptReadData   := ADR(zz_DataField_1_Read);

(*----------------------------------------------------*)


(*#### START OF FIXED CODE #####################################*)
zz_MBCFG_MASTER_ETH(	strIpAddress    := MBCFG_IpAddress,                 (* fixed entry     *)
                        uiPort          := MBCFG_Port,                      (* fixed entry     *)
                        bUnitID         := MBCFG_UnitID,                    (* fixed entry     *)
                        tTimeOut        := MBCFG_TimeOut,                   (* fixed entry     *)
                        iVariableCount  := zz_VARIABLECOUNT,
                        ptVariableList  := ADR(zz_VariableList),
                        iJobCount       := zz_JOBCOUNT,
                        ptJobList       := ADR(zz_JobList),
                        tRequestDelay   := MBCFG_RequestDelay,              (* fixed entry     *)
                        eError          => MBCFG_Error,                     (* fixed entry     *)
                        LastJob         => MBCFG_LastJob                    (* fixed entry     *)
                    );
(*##############################################################*)
END_PROGRAM

(* POU SWD, ST *)
FUNCTION_BLOCK SWD
VAR_INPUT
END_VAR
VAR_OUTPUT
END_VAR
VAR
END_VAR
   (*SWD_swd_ctr_mode_0 AT %QW271: UINT;*)
IF           H_AT_SEA = TRUE       THEN  SWD_swd_ctr_mode_0:=1;(*AT SEA*)
ELSIF    H_STAND_BY = TRUE  THEN  SWD_swd_ctr_mode_0:=2;(*STAND BY*)
ELSIF    H_FINSHED_WITH_ENGINE     THEN  SWD_swd_ctr_mode_0:=3;(*FWE *)
ELSE  SWD_swd_ctr_mode_0:=0;(* UKN*)
END_IF;
END_FUNCTION_BLOCK

(* POU OutputProgramValueMapping, ST *)
FUNCTION_BLOCK OutputProgramValueMapping
VAR_INPUT
END_VAR
VAR_OUTPUT
END_VAR
VAR
END_VAR
(***************Bridge_Control_Position_Change***************)
BR_CENTRL_PORT_CONTROL_IN_CONTROL := BRIDGE_PORT_EOT_IN_CONTROL_LAMP;(*PROEOT1043*)
BR_CENTRL_STBD_CONTROL_IN_CONTROL := BRIDGE_STBD_EOT_IN_CONTROL_LAMP;(*PROEOT1044*)
BR_PORT_CONTROL_IN_CONTROL := PORT_EOT_IN_CONTROL_LAMP
										   OR  PORT_LAMP_TEST_PB;(*PROEOT1045*)
BR_STBD_CONTROL_IN_CONTROL := STBD_EOT_IN_CONTROL_LAMP
									      	   OR  STBD_LAMP_TEST_PB;(*PROEOT1046*)

(*PORT or  STBD in control*)
HW_PORT_IN_CONTROL := BRG_PORT_IN_CONTROL;
HW_STBD_IN_CONTROL := BRG_STBD_IN_CONTROL;


(*HMI*)
H_PORT_WING_CONTRL := BRG_PORT_IN_CONTROL;(*PROEOT0007*)
H_STBD_WING_CONTRL := BRG_STBD_IN_CONTROL;(*PROEOT0008*)

(***************MVL***************)
(*indicator*)
BR_Indicator_Position_Pointer := BR_Indicator_Position_Pointer_P;(*PROEOT1006*)
PORT_BR_Indicator_Position_Pointer := BR_PORT_Indicator_Position_Pointer_P;(*PROEOT1011*)
STBD_BR_Indicator_Position_Pointer := BR_STBD_Indicator_Position_Pointer_P;(*PROEOT1012*)
ECR_Indicator_Position_Pointer := ECR_Indicator_Position_Pointer_P;(*PROEOT1008*)
LOCAL_Indicator_Position_Pointer := LOCAL_Indicator_Position_Pointer_P;(*PROEOT1010*)

(********TEST********)
TEST_LOCAL_Telegraph_Position_Pointer  := TEST_LOCAL_Telegraph_Position_Pointer_P;

(*LOCAL MAN CTRL*)
LOCAL_IN_CONTROL_TAKE_ON_INDICATOR := LOCAL_MAN_CTRL;(*PROEOT1047*)
(*hmi*)
LOCAL_MAN_TAKE_OVER := LOCAL_IN_CONTROL_TAKE_ON_INDICATOR;

(*HMI--------POWER LOST*)
(*OR  LAMP TEST PB*)
H_ECR_TElegraph_POWER_LOST := ECR_TElegraph_POWER_LOST_P  OR  LAMP_TEST_PB;(*PROEOT0009*)
H_LOCAL_TElegraph_POWER_LOST := LOCAL_TElegraph_POWER_LOST_P  OR  LAMP_TEST_PB; (*PROEOT0010*)
H_PORT_TElegraph_POWER_LOST := PORT_TElegraph_POWER_LOST_P  OR  LAMP_TEST_PB; (*PROEOT0011*)
H_STBD_TElegraph_POWER_LOST := STBD_TElegraph_POWER_LOST_P  OR  LAMP_TEST_PB; (*PROEOT0012*)
H_BR_TElegraph_POWER_LOST := BR_TElegraph_POWER_LOST_P  OR  LAMP_TEST_PB; (*PROEOT0013*)


TELEGRAPH_SUB_SYS_PWR_LOST_MBO :=	TELEGRAPH_SUB_SYS_PWR_LOST;

(***************Sub_telegraph_function***************)
STANDBY_BR_INDICATOR := INDICATOR_STANDBY_BRG  OR  BR_LAMP_TEST_PB;(*PROEOT1029*)
AT_SEA_BR_PB_INDICATOR := INDICATOR_ATSEA_BRG  OR  BR_LAMP_TEST_PB;(*PROEOT1030*)
FWE_BR_PB_INDICATOR := INDICATOR_FWE_BRG  OR  BR_LAMP_TEST_PB;(*PROEOT1031*)

STANDBY_ECR_AUT_PB_INDICATOR := INDICATOR_STANDBY_MCR  OR  ECR_LAMP_TEST_PB;(*PROEOT1033*)
AT_SEA_ECR_AUT_PB_INDICATOR := INDICATOR_ATSEA_MCR  OR  ECR_LAMP_TEST_PB;(*PROEOT1034*)
FWE_ECR_AUT_PB_INDICATOR := INDICATOR_FWE_MCR  OR  ECR_LAMP_TEST_PB;(*PROEOT1035*)

STANDBY_LOCAL_INDICATOR := INDICATOR_STANDBY_LC;(*PROEOT1037*)
AT_SEA_LOCAL_INDICATOR := INDICATOR_ATSEA_LC;(*PROEOT1038*)
FWE_LOCAL_INDICATOR := INDICATOR_FWE_LC;(*PROEOT1039*)

(***************WRONG WAY******************)
(*HW*)
HW_WRONG_WAY_BR :=  WRONG_WAY
						OR  BRIDGE_LAMP_TEST_PB;

HW_WRONG_WAY_ECR :=  WRONG_WAY
						OR  ECR_LAMP_TEST_PB;
(*HMI*)
H_WRONG_WAY := WRONG_WAY
						OR  LAMP_TEST_PB;


(***************Mismatch Alarm***************)
BR_TELEGRAPH_ORDER_Acoustic_Signal :=( BRG_CENR_IN_CONTROL AND (TELEGRAPH_ORDER_BR
													 OR WRONG_WAY
													 OR  BUZZER_BRG
													 OR BRIDGE_BUZZER
													OR FRM_FAIL_ACOUSTIC_BUZZER) ) OR BR_LAMP_TEST_PB OR FRM_CONTROL_TRANS_BUZZER_BRG;

PORT_TELEGRAPH_ORDER_Acoustic_Signal :=(BRG_PORT_IN_CONTROL AND ( TELEGRAPH_ORDER_PORT
													 OR  PORT_BUZZER
													OR FRM_FAIL_ACOUSTIC_BUZZER ) ) OR  PORT_LAMP_TEST_PB OR FRM_CONTROL_TRANS_BUZZER_BRG;

STBD_TELEGRAPH_ORDER_Acoustic_Signal := (BRG_STBD_IN_CONTROL AND (TELEGRAPH_ORDER_STBD
													 OR  STBD_BUZZER
													OR  FRM_FAIL_ACOUSTIC_BUZZER )  )  OR  STBD_LAMP_TEST_PB OR FRM_CONTROL_TRANS_BUZZER_BRG ;

ECR_TELEGRAPH_ORDER_Acoustic_Signal :=( (FRM_ECR_AUT_CONTROL OR FRM_ECR_MAN_CONTROL) AND ((TELEGRAPH_ORDER_ECR AND NOT FRM_ECR_MAN_CONTROL)
													OR WRONG_WAY
													OR  BUZZER_MCR
													OR FRM_FAIL_ACOUSTIC_BUZZER)) OR  ECR_LAMP_TEST_PB OR FRM_CONTROL_TRANS_BUZZER_MCR;
LOCAL_TELEGRAPH_ORDER_Acoustic_Signal := TELEGRAPH_ORDER_LC
													OR WRONG_WAY;

(*HMI*)
H_TELEGRAPH_COINCIDENCE := TELEGRAPH_COINCIDENCE;(*PROEOT0006*)
TELEGRAPH_HORN_ALARM_MBO := TELEGRAPH_ORDER_ECR;

(***************EOT_system_failure_Alarm***************)
Telegraph_System_Failure_ALM := TELEGRAPH_SYSTEM_FAIL_XS9021A;(*PROEOTXS9021A*)


(*HMI*)
H_BR_TElegraph_PASSIVE_FAIL := PASSIVE_FAILURE_BR
										OR  LAMP_TEST_PB;(*PROEOT0034*)
H_ECR_TElegraph_PASSIVE_FAIL := PASSIVE_FAILURE_ECR
										OR  LAMP_TEST_PB;(*PROEOT0035*)
H_LOCAL_TElegraph_PASSIVE_FAIL := PASSIVE_FAILURE_LC
										OR  LAMP_TEST_PB;(*PROEOT0036*)
H_PORT_TElegraph_PASSIVE_FAIL := PASSIVE_FAILURE_BR_PORT
										OR  LAMP_TEST_PB; (*PROEOT0037*)
H_STBD_TElegraph_PASSIVE_FAIL := PASSIVE_FAILURE_BR_STBD
										OR  LAMP_TEST_PB;(*PROEOT0038*)

TELEGRAPH_SYS_PASS_FAIL_9021A_MBO :=  TELEGRAPH_SYSTEM_FAIL_XS9021A;

(***************AMPERE_STAGE_TO_HMI***************)
Telegraph_Indicator_Full_SEA_AH_MBO := Telegraph_Indicator_Full_SEA_AH;
Telegraph_Indicator_FULL_AH_MBO := Telegraph_Indicator_FULL_AH;
Telegraph_Indicator_HALF_AH_MBO := Telegraph_Indicator_HALF_AH;
Telegraph_Indicator_SLOW_AH_MBO := Telegraph_Indicator_SLOW_AH;
Telegraph_Indicator_DEAD_S_AH_MBO := Telegraph_Indicator_DEAD_S_AH;
Telegraph_Indicator_STOP_MBO := Telegraph_Indicator_STOP;
Telegraph_Indicator_DEAD_S_AS_MBO := Telegraph_Indicator_DEAD_S_AS;
Telegraph_Indicator_SLOW_AS_MBO := Telegraph_Indicator_SLOW_AS;
Telegraph_Indicator_HALF_AS_MBO := Telegraph_Indicator_HALF_AS;
Telegraph_Indicator_FULL_AS_MBO := Telegraph_Indicator_FULL_AS;
Telegraph_Indicator_Emergency_AS_MBO := Telegraph_Indicator_Emergency_AS;


(***************MVL_COMMD_TO_RCS***************)
(*TO RCS*)
ECR_MVL_COMMD_TO_RCS := ECR_MVL_COMMD_TO_RCS_P;(*PROEOT1009*)
BR_MVL_COMMD_TO_RCS := BR_MVL_COMMD_TO_RCS_P; (*PROEOT1007*)
END_FUNCTION_BLOCK

(* POU WRONG_WAY, ST *)
(*4.1.7.1.3*)
FUNCTION_BLOCK WRONG_WAY
VAR_INPUT
END_VAR
VAR_OUTPUT

END_VAR
VAR
	TON_WORNG_WAY: TON;
	TEMP_WRONG_WAY: BOOL;
END_VAR
(*4.1.7.1.3*)
(*GET MVL POSITION AHEAD AND ASTERN*)
(*AHEAD*)
IF    (Telegraph_Indicator_Full_SEA_AH
	OR	Telegraph_Indicator_FULL_AH
	OR Telegraph_Indicator_HALF_AH
	OR Telegraph_Indicator_SLOW_AH
	OR Telegraph_Indicator_DEAD_S_AH)
THEN
	MVL_POSITION_AHEAD := TRUE;
	MVL_POSITION_ASTERN := FALSE;
(*ASTERN*)
ELSIF  (Telegraph_Indicator_DEAD_S_AS
		OR Telegraph_Indicator_SLOW_AS
		OR Telegraph_Indicator_HALF_AS
		OR Telegraph_Indicator_FULL_AS
		OR Telegraph_Indicator_Emergency_AS)
THEN
	MVL_POSITION_AHEAD := FALSE;
	MVL_POSITION_ASTERN := TRUE;
(*STOP*)
ELSE
	MVL_POSITION_AHEAD := FALSE;
	MVL_POSITION_ASTERN := FALSE;
END_IF


(*GET ENG TURN AHEAD OR ASTERN*)
(*
ENGINE_TURN_AHEAD := (FRM_ENG_TURNING_AHEAD AND NOT FRM_ENG_SENSOR_1_FAILURE)
							OR (ESS_ENG_TURNING_AHEAD AND NOT ESS_ENG_SENSOR_1_FAILURE);

ENGINE_TURN_ASTERN := (FRM_ENG_TURNING_AST AND NOT FRM_ENG_SENSOR_1_FAILURE)
							 OR (ESS_ENG_TURNING_AST AND NOT ESS_ENG_SENSOR_1_FAILURE);
*)
ENGINE_TURN_AHEAD :=	ESS_ENG_TURNING_AHEAD AND NOT ESS_ENG_SENSOR_1_FAILURE;
ENGINE_TURN_ASTERN :=	ESS_ENG_TURNING_AST AND NOT ESS_ENG_SENSOR_1_FAILURE;

(*GET MCR CONTROL*)
MCR_LC_CONTROL := ECR_MAN_CONTROL
					OR LOCAL_MAN_CTRL;

(****WRONG WAY ALARM****)
TEMP_WRONG_WAY := MCR_LC_CONTROL
					AND ((MVL_POSITION_AHEAD AND ENGINE_TURN_ASTERN) OR (MVL_POSITION_ASTERN AND ENGINE_TURN_AHEAD));

TON_WORNG_WAY(IN := TEMP_WRONG_WAY, PT := T#5S);

WRONG_WAY := TON_WORNG_WAY.Q;
END_FUNCTION_BLOCK

(* POU MVL_COMMAND, ST *)
(*4.1.7.1.1*)
FUNCTION_BLOCK MVL_COMMAND
VAR_INPUT
END_VAR
VAR_OUTPUT
END_VAR
VAR
	Bridge_Control_Position_Change_FUNC: Bridge_Control_Position_Change;

	InputCut1 : REAL;
	InputCut2 : REAL;
	InputCut3 : REAL;

END_VAR
(*GET   Control Position in BRIDGE*)
Bridge_Control_Position_Change_FUNC;

(***********GET TELEGRAPH_POSITION_BR****************)

IF  BRG_CENR_IN_CONTROL = TRUE
THEN
	TELEGRAPH_POSITION_BR :=  CENT_EOT_MVL;
ELSIF  BRG_PORT_IN_CONTROL = TRUE
THEN
	TELEGRAPH_POSITION_BR :=  PORT_WING_EOT_MVL;
ELSIF	BRG_STBD_IN_CONTROL = TRUE
THEN
	TELEGRAPH_POSITION_BR := STBD_WING_EOT_MVL;
ELSE
	TELEGRAPH_POSITION_BR :=  CENT_EOT_MVL;
END_IF

(*test  4~20mA*)
InputCut1 := WORD_TO_REAL( CENT_EOT_MVL ) /  AD_Scale;
InputCut2 := WORD_TO_REAL( ECR_MVL_COMMD ) /  AD_Scale;
InputCut3 := WORD_TO_REAL (LOCAL_MVL_COMMD) /  AD_Scale;


(*4.1.7.1.1*)
(********************MVL COMMAND***********************)

TELEGRAPH_INDICATOR_ECR := TELEGRAPH_POSITION_BR;(*BR_MVL_COMMD*)
TELEGRAPH_INDICATOR_LC := TELEGRAPH_POSITION_BR;

(*TELEGRAPH_INDICATOR_BR*)
IF LOCAL_MAN_CTRL = TRUE
THEN
	TELEGRAPH_INDICATOR_BR := TELEGRAPH_POSITION_LC;
ELSE
	IF (ECR_AUT_CTRL OR ECR_MAN_CONTROL) = TRUE
	THEN
		TELEGRAPH_INDICATOR_BR := TELEGRAPH_POSITION_CR;
	ELSE
		TELEGRAPH_INDICATOR_BR := TELEGRAPH_POSITION_BR;
	END_IF
END_IF

TELEGRAPH_INDICATOR_BR_PORT := TELEGRAPH_INDICATOR_BR;
TELEGRAPH_INDICATOR_BR_STBD := TELEGRAPH_INDICATOR_BR;

(***************MVL POWER LOST****************)
(*
H_ECR_TElegraph_POWER_LOST := ECR_TElegraph_POWER_LOST_P;(*PROEOT0009*)
H_LOCAL_TElegraph_POWER_LOST := LOCAL_TElegraph_POWER_LOST_P; (*PROEOT0010*)
H_PORT_TElegraph_POWER_LOST := PORT_TElegraph_POWER_LOST_P; (*PROEOT0011*)
H_STBD_TElegraph_POWER_LOST := STBD_TElegraph_POWER_LOST_P; (*PROEOT0012*)
H_BR_TElegraph_POWER_LOST := BR_TElegraph_POWER_LOST_P; (*PROEOT0013*)
*)

(*HMI*)
TELEGRAPH_SUB_SYS_PWR_LOST :=	ECR_TElegraph_POWER_LOST_P
												OR  LOCAL_TElegraph_POWER_LOST_P
												OR  PORT_TElegraph_POWER_LOST_P
												OR  STBD_TElegraph_POWER_LOST_P
												OR  BR_TElegraph_POWER_LOST_P;
END_FUNCTION_BLOCK

(* POU Bridge_Control_Position_Change, ST *)
FUNCTION_BLOCK Bridge_Control_Position_Change
VAR_INPUT
END_VAR
VAR_OUTPUT
END_VAR
VAR
	BLINK_LAMP: BLINK;
	BLINK_TIME: TIME;

	(*MVL不匹配误差 暂定2MA*)
	MVL_MISMATCH_TEMP: WORD;


	(*transfer process  time out*)
	TON_TIMEOUT: TON;
	(*transfer of TAKE process timer*)
	TON_TAKE: TON;

	(*waiting for STBD , PORT confirm   flag*)
	BR_CENR_SUPPLY_TO_PORT_REQUEST: BOOL := FALSE;
	BR_CENR_SUPPLY_TO_STBD_REQUEST: BOOL := FALSE;

	BR_CENR_TAKE_FROM_PORT_REQUEST: BOOL := FALSE;
	BR_CENR_TAKE_FROM_STBD_REQUEST: BOOL := FALSE;

	(*in change process  flag *)
	CENR_SUPPLY_TO_PORT_IN_PROCESS: BOOL := FALSE;
	CENR_SUPPLY_TO_STBD_IN_PROCESS: BOOL := FALSE;

	CENR_TAKE_FROM_PORT_IN_PROCESS: BOOL := FALSE;
	CENR_TAKE_FROM_STBD_IN_PROCESS: BOOL := FALSE;

END_VAR
(*if port or stbd is in control, the telegraph indicator should be showing the current command*)
(*BR_Telegraph_Position_Pointer   PORT_BR_Telegraph_Position_Pointer   STBD_BR_Telegraph_Position_Pointer*)


(*****init  bridge lamp status, default control in CENTER******)
IF	CONTROL_TRANS_PROCESS_FLAG = FALSE
THEN
	IF	BRG_CENR_IN_CONTROL = TRUE
	THEN
		(*ALL lamp keep off*)
		BRIDGE_PORT_EOT_IN_CONTROL_LAMP := FALSE;
		BRIDGE_STBD_EOT_IN_CONTROL_LAMP := FALSE;
		PORT_EOT_IN_CONTROL_LAMP := FALSE;
		STBD_EOT_IN_CONTROL_LAMP := FALSE;
	ELSIF  BRG_STBD_IN_CONTROL = TRUE
	THEN
		(*LAMP*)
		BRIDGE_PORT_EOT_IN_CONTROL_LAMP := FALSE;
		BRIDGE_STBD_EOT_IN_CONTROL_LAMP := TRUE;
		PORT_EOT_IN_CONTROL_LAMP := FALSE;
		STBD_EOT_IN_CONTROL_LAMP := TRUE;
	ELSIF  BRG_PORT_IN_CONTROL = TRUE
	THEN
		(*LAMP*)
		BRIDGE_PORT_EOT_IN_CONTROL_LAMP := TRUE;
		BRIDGE_STBD_EOT_IN_CONTROL_LAMP := FALSE;
		PORT_EOT_IN_CONTROL_LAMP := TRUE;
		STBD_EOT_IN_CONTROL_LAMP := FALSE;
	END_IF
END_IF



IF BRG_IN_CONTROL_P = FALSE
	AND  CONTROL_TRANS_PROCESS_FLAG = FALSE
THEN
	RETURN;
END_IF


(*LMAP BLINK*)
(*
BLINK_TIME := REAL_TO_TIME((1.0/Flasher_frequency_P) * 0.5);
BLINK_LAMP(ENABLE := TRUE, TIMELOW :=BLINK_TIME, TIMEHIGH :=BLINK_TIME);
*)
IF  Flasher_frequency_P >= 0.5
	AND  Flasher_frequency_P < 0.75
THEN
	(*frequency set 0.5Hz*)
	BLINK_TIME := t#1s;
ELSIF	Flasher_frequency_P >= 0.75
		AND Flasher_frequency_P <= 1.25
THEN
	(*frequency set 1Hz*)
	BLINK_TIME := t#0.5s;
ELSIF	Flasher_frequency_P > 1.25
		AND Flasher_frequency_P <= 1.75
THEN
	(*frequency set 1.5hz*)
	BLINK_TIME := t#0.33s;
ELSIF	Flasher_frequency_P > 1.75
		AND Flasher_frequency_P <= 2
THEN
	(*frequency set 2hz*)
	BLINK_TIME := t#0.25s;
ELSE
	(*frequency set 0.5hz*)
	BLINK_TIME := t#1s;
END_IF

BLINK_LAMP(ENABLE := TRUE, TIMELOW :=BLINK_TIME, TIMEHIGH :=BLINK_TIME);


MVL_MISMATCH_TEMP := 2 * AD_SCALE;

(*********control transfer between WING EOTs and BRG CENR EOT***********************)

(******control transfer between PORT and CENTER***********)
(*--------------------------SUPPLY  PORT--------------------------*)
IF PORT_BUTTON_EOT_IN_CNTR = TRUE
THEN
	(*if not during transfer process and control in center*)
	IF  BRG_CENR_IN_CONTROL = TRUE
		AND CONTROL_TRANS_PROCESS_FLAG = FALSE
	THEN
		(*set during transfer process*)
		CONTROL_TRANS_PROCESS_FLAG := TRUE;
		(*CENTER  supply  to  PORT process flag  set  TRUE*)
		CENR_SUPPLY_TO_PORT_IN_PROCESS := TRUE;
	END_IF
END_IF

(*in process*)
IF	CENR_SUPPLY_TO_PORT_IN_PROCESS = TRUE
THEN
	(*start timeout exit timer*)
	TON_TIMEOUT(IN := TRUE, PT := t#30s);
	(*lamp of PORT and CENTER flick*)
	PORT_EOT_IN_CONTROL_LAMP := BLINK_LAMP.OUT;
	BRIDGE_PORT_EOT_IN_CONTROL_LAMP := BLINK_LAMP.OUT; (*****)
	(*PORT BUZZER active*)
	PORT_BUZZER := TRUE;

	(*if MVL COMMAND  dont match*)
	IF	ABS(PORT_WING_EOT_MVL - CENT_EOT_MVL) > MVL_MISMATCH_TEMP
	THEN
		(*waiting for PORT WING confirm and set request flag false,means ignor the PORT confirm button*)
		BR_CENR_SUPPLY_TO_PORT_REQUEST := FALSE;
		(*CENTER BUZZER active*)
		BRIDGE_BUZZER := TRUE;
	ELSE
		(*waiting for PORT WING confirm and set request flag true*)
		BR_CENR_SUPPLY_TO_PORT_REQUEST := TRUE;
		(*CENTER BUZZER silence*)
		BRIDGE_BUZZER := FALSE;
	END_IF
END_IF


(*waiting for PORT WING confirm*)
IF	BR_CENR_SUPPLY_TO_PORT_REQUEST = TRUE
THEN
	IF	PORT_BUTTON_EOT = TRUE
	THEN
		(*transfer available to PORT*)
		BRG_PORT_IN_CONTROL := TRUE;
		BRG_CENR_IN_CONTROL := FALSE;
		BRG_STBD_IN_CONTROL := FALSE;
		(*port wing  and CENTER  lamp turn on*)
		PORT_EOT_IN_CONTROL_LAMP := TRUE;
		BRIDGE_PORT_EOT_IN_CONTROL_LAMP := TRUE;
		BRIDGE_STBD_EOT_IN_CONTROL_LAMP := FALSE;
		STBD_EOT_IN_CONTROL_LAMP := FALSE;
		(*PORT BUZZER SILENCE*)
		PORT_BUZZER := FALSE;
		(*transfer process down*)
		CONTROL_TRANS_PROCESS_FLAG := FALSE;
		(*request flag set false*)
		BR_CENR_SUPPLY_TO_PORT_REQUEST := FALSE;
		(*CENTER  supply  to  PORT process flag  set  FALSE*)
		CENR_SUPPLY_TO_PORT_IN_PROCESS := FALSE;
		(*stop  time out timer*)
		TON_TIMEOUT(IN := FALSE);
	END_IF
END_IF

(*--------------------------TAKE PORT-------------------------------*)
IF PORT_BUTTON_EOT_IN_CNTR = TRUE
THEN
	(*if not during transfer process and control in PORT*)
	IF  BRG_PORT_IN_CONTROL = TRUE
		AND CONTROL_TRANS_PROCESS_FLAG = FALSE
	THEN
		(*set during transfer process*)
		CONTROL_TRANS_PROCESS_FLAG := TRUE;
		(*CENTER  TAKE  FROM  PORT process flag  set  TRUE*)
		CENR_TAKE_FROM_PORT_IN_PROCESS := TRUE;
	END_IF
END_IF

IF	CENR_TAKE_FROM_PORT_IN_PROCESS = TRUE
THEN
	(*start timeout exit timer*)
	TON_TIMEOUT(IN := TRUE, PT := t#30s);

	(*if MVL COMMAND  dont match*)
	IF	ABS(PORT_WING_EOT_MVL - CENT_EOT_MVL) > MVL_MISMATCH_TEMP
	THEN
		(*center lamp flick, port lamp keep on*)
		BRIDGE_PORT_EOT_IN_CONTROL_LAMP := BLINK_LAMP.OUT;
		PORT_EOT_IN_CONTROL_LAMP := TRUE;
	ELSE
		(***MVL COMMAND  match***)
		(*transfer available to CENTER*)
		BRG_PORT_IN_CONTROL := FALSE;
		BRG_CENR_IN_CONTROL := TRUE;
		BRG_STBD_IN_CONTROL := FALSE;
		(*start TAKE process DELAY  2S*)
		TON_TAKE(IN := TRUE, PT := t#2s);
		(*CENTER IN control*)
		(*LAMP in CENTER and PORT turn off*)
		BRIDGE_PORT_EOT_IN_CONTROL_LAMP := FALSE;
		PORT_EOT_IN_CONTROL_LAMP := FALSE;
		(*BUZZER in CENTER and PORT turn ON*)
		BRIDGE_BUZZER := TRUE;
		PORT_BUZZER := TRUE;
		(*STOP  timeout  timer*)
		TON_TIMEOUT(IN := FALSE);
		(*TAKE PORT WING request flag set  true*)
		BR_CENR_TAKE_FROM_PORT_REQUEST := TRUE;
	END_IF
END_IF

(**wait for TAKE time out, means the TAKE control process completed**)
IF  TON_TAKE.Q = TRUE
	AND BR_CENR_TAKE_FROM_PORT_REQUEST = TRUE
THEN
	(*PORT and CENTER BUZZER SILENCE*)
	BRIDGE_BUZZER := FALSE;
	PORT_BUZZER := FALSE;
	(*transfer process down*)
	CONTROL_TRANS_PROCESS_FLAG := FALSE;
	(*TAKE PORT WING request flag set  FALSE*)
	BR_CENR_TAKE_FROM_PORT_REQUEST := FALSE;
	(*STOP TAKE timer *)
	TON_TAKE(IN := FALSE);
	CENR_TAKE_FROM_PORT_IN_PROCESS := FALSE;
END_IF


(******control transfer between STBD and CENTER******)
(*--------------------------SUPPLY		STBD--------------------------*)
IF STBD_BUTTON_EOT_IN_CNTR = TRUE
THEN
	(*if not during transfer process and control in center*)
	IF  BRG_CENR_IN_CONTROL = TRUE
		AND CONTROL_TRANS_PROCESS_FLAG = FALSE
	THEN
		(*set during transfer process*)
		CONTROL_TRANS_PROCESS_FLAG := TRUE;
		CENR_SUPPLY_TO_STBD_IN_PROCESS := TRUE;
	END_IF
END_IF

IF	CENR_SUPPLY_TO_STBD_IN_PROCESS = TRUE
THEN
	(*start timeout exit timer*)
	TON_TIMEOUT(IN := TRUE, PT := t#30s);
	(*lamp of STBD and CENTER flick*)
	STBD_EOT_IN_CONTROL_LAMP := BLINK_LAMP.OUT;
	BRIDGE_STBD_EOT_IN_CONTROL_LAMP := BLINK_LAMP.OUT;
	(*STBD BUZZER active*)
	STBD_BUZZER := TRUE;

	(*if MVL COMMAND  dont match*)
	IF	ABS(STBD_WING_EOT_MVL - CENT_EOT_MVL) > MVL_MISMATCH_TEMP
	THEN
		(*waiting for STBD WING confirm set request flag false,means ignor the STBD confirm button*)
		BR_CENR_SUPPLY_TO_STBD_REQUEST := FALSE;
		(*CENTER BUZZER active*)
		BRIDGE_BUZZER := TRUE;
	ELSE
		(*waiting for STBD WING confirm and set request flag true*)
		BR_CENR_SUPPLY_TO_STBD_REQUEST := TRUE;
		(*CENTER BUZZER silence*)
		BRIDGE_BUZZER := FALSE;
	END_IF
END_IF

(*waiting for STBD WING confirm*)
IF	BR_CENR_SUPPLY_TO_STBD_REQUEST = TRUE
THEN
	IF	STBD_BUTTON_EOT = TRUE
	THEN
		(*transfer available to STBD*)
		BRG_PORT_IN_CONTROL := FALSE;
		BRG_CENR_IN_CONTROL := FALSE;
		BRG_STBD_IN_CONTROL := TRUE;
		(*bridge control indicator off*)
		(*STBD wing  and CENTER  lamp turn on*)
		PORT_EOT_IN_CONTROL_LAMP := FALSE;
		BRIDGE_STBD_EOT_IN_CONTROL_LAMP := TRUE;
		STBD_EOT_IN_CONTROL_LAMP := TRUE;
		(*STBD BUZZER SILENCE*)
		STBD_BUZZER := FALSE;
		(*transfer process down*)
		CONTROL_TRANS_PROCESS_FLAG := FALSE;
		(*request flag set false*)
		BR_CENR_SUPPLY_TO_STBD_REQUEST := FALSE;
		CENR_SUPPLY_TO_STBD_IN_PROCESS := FALSE;
		(*stop  time out timer*)
		TON_TIMEOUT(IN := FALSE);
	END_IF
END_IF

(*--------------------------TAKE STBD-------------------------------*)
IF STBD_BUTTON_EOT_IN_CNTR = TRUE
THEN
	(*if not during transfer process and control in STBD*)
	IF  BRG_STBD_IN_CONTROL = TRUE
		AND CONTROL_TRANS_PROCESS_FLAG = FALSE
	THEN
		(*set during transfer process*)
		CONTROL_TRANS_PROCESS_FLAG := TRUE;
		CENR_TAKE_FROM_STBD_IN_PROCESS := TRUE;
	END_IF
END_IF

IF	CENR_TAKE_FROM_STBD_IN_PROCESS = TRUE
THEN
	(*start timeout exit timer*)
	TON_TIMEOUT(IN := TRUE, PT := t#30s);

	(*if MVL COMMAND  dont match*)
	IF	ABS(STBD_WING_EOT_MVL - CENT_EOT_MVL) > MVL_MISMATCH_TEMP
	THEN
		(*center lamp flick, STBD lamp keep on*)
		BRIDGE_STBD_EOT_IN_CONTROL_LAMP := BLINK_LAMP.OUT;
		STBD_EOT_IN_CONTROL_LAMP := TRUE;
	ELSE
		(***MVL COMMAND  match***)
		(*transfer available to PORT*)
		BRG_PORT_IN_CONTROL := FALSE;
		BRG_CENR_IN_CONTROL := TRUE;
		BRG_STBD_IN_CONTROL := FALSE;
		(*start TAKE process DELAY  2S*)
		TON_TAKE(IN := TRUE, PT := t#2s);
		(*CONTROL in center*)
		(*LAMP in CENTER and STBD turn off*)
		BRIDGE_STBD_EOT_IN_CONTROL_LAMP := FALSE;
		STBD_EOT_IN_CONTROL_LAMP := FALSE;
		(*BUZZER in CENTER and STBD turn ON*)
		BRIDGE_BUZZER := TRUE;
		STBD_BUZZER := TRUE;
		(*STOP  timeout  timer*)
		TON_TIMEOUT(IN := FALSE);
		(*TAKE PORT WING request flag set  true*)
		BR_CENR_TAKE_FROM_STBD_REQUEST := TRUE;
	END_IF
END_IF

(**wait for TAKE time out, means the TAKE control process completed**)
IF  TON_TAKE.Q = TRUE
	AND BR_CENR_TAKE_FROM_STBD_REQUEST = TRUE
THEN
	(*STBD and CENTER BUZZER SILENCE*)
	BRIDGE_BUZZER := FALSE;
	STBD_BUZZER := FALSE;
	(*transfer process down*)
	CONTROL_TRANS_PROCESS_FLAG := FALSE;
	(*TAKE STBD WING request flag set  FALSE*)
	BR_CENR_TAKE_FROM_STBD_REQUEST := FALSE;
	CENR_TAKE_FROM_STBD_IN_PROCESS := FALSE;
	(*STOP TAKE timer *)
	TON_TAKE(IN := FALSE);
END_IF



(****timer out process****)
IF	TON_TIMEOUT.Q = TRUE
	AND CONTROL_TRANS_PROCESS_FLAG = TRUE
THEN
	(*all the request flag  set false*)
	CONTROL_TRANS_PROCESS_FLAG := FALSE;

	BR_CENR_SUPPLY_TO_PORT_REQUEST := FALSE;
	BR_CENR_SUPPLY_TO_STBD_REQUEST := FALSE;
	BR_CENR_TAKE_FROM_PORT_REQUEST  := FALSE;
	BR_CENR_TAKE_FROM_STBD_REQUEST  := FALSE;

	CENR_SUPPLY_TO_PORT_IN_PROCESS := FALSE;
	CENR_SUPPLY_TO_STBD_IN_PROCESS := FALSE;
	CENR_TAKE_FROM_PORT_IN_PROCESS := FALSE;
	CENR_TAKE_FROM_STBD_IN_PROCESS := FALSE;

	(*RESET transfer process*)
	(*all buzzer silience*)
	BRIDGE_BUZZER := FALSE;
	PORT_BUZZER := FALSE;
	STBD_BUZZER := FALSE;

	IF	BRG_CENR_IN_CONTROL = TRUE
	THEN
		(*ALL lamp keep off*)
		BRIDGE_PORT_EOT_IN_CONTROL_LAMP := FALSE;
		BRIDGE_STBD_EOT_IN_CONTROL_LAMP := FALSE;
		PORT_EOT_IN_CONTROL_LAMP := FALSE;
		STBD_EOT_IN_CONTROL_LAMP := FALSE;
	ELSIF  BRG_STBD_IN_CONTROL = TRUE
	THEN
		(*LAMP*)
		BRIDGE_PORT_EOT_IN_CONTROL_LAMP := FALSE;
		BRIDGE_STBD_EOT_IN_CONTROL_LAMP := TRUE;
		PORT_EOT_IN_CONTROL_LAMP := FALSE;
		STBD_EOT_IN_CONTROL_LAMP := TRUE;
	ELSIF  BRG_PORT_IN_CONTROL = TRUE
	THEN
		(*LAMP*)
		BRIDGE_PORT_EOT_IN_CONTROL_LAMP := TRUE;
		BRIDGE_STBD_EOT_IN_CONTROL_LAMP := FALSE;
		PORT_EOT_IN_CONTROL_LAMP := TRUE;
		STBD_EOT_IN_CONTROL_LAMP := FALSE;
	END_IF
	(*time out timer stop*)
	TON_TIMEOUT(IN := FALSE);
END_IF
END_FUNCTION_BLOCK

(* POU Sub_telegraph_function, ST *)
(*4.1.7.1.2*)
FUNCTION_BLOCK Sub_telegraph_function
VAR_INPUT
END_VAR
VAR_OUTPUT
END_VAR
VAR
	INDICATOR_FLASH: BLINK;
	TON_TIMEOUT: TON;
	(*FWE status delay timer*)
	TON_FWE_TIMER: TON;

	(*the pushbutton pressed flag from BRG,MCR, not pressed = FALSE,  pressed = TRUE*)
	BRG_STANDBY_PRESSED_FLAG: BOOL := FALSE;
	MCR_STANDBY_PRESSED_FLAG: BOOL := FALSE;

	BRG_ATSEA_PRESSED_FLAG: BOOL := FALSE;
	MCR_ATSEA_PRESSED_FLAG: BOOL := FALSE;

	BRG_FWE_PRESSED_FLAG: BOOL := FALSE;
	MCR_FWE_PRESSED_FLAG: BOOL := FALSE;

	(*the MCR pushbutton already pressed firest time flag*)
	MCR_STANDBY_FST_PRESSED_FLAG: BOOL := FALSE;
	MCR_ATSEA_FST_PRESSED_FLAG: BOOL := FALSE;
	MCR_FWE_FST_PRESSED_FLAG: BOOL := FALSE;

	(*in  process flag*)
	STANDBY_IN_PROCESS_FLAG: BOOL := FALSE;
	ATSEA_IN_PROCESS_FLAG: BOOL := FALSE;
	FWE_IN_PROCESS_FLAG: BOOL := FALSE;

	(*indicator flash flag*)
	STANDBY_PRO_IND_FLASH_FLAG: BOOL := FALSE;
	ATSEA_PRO_IND_FLASH_FLAG: BOOL := FALSE;
	FWE_PRO_IND_FLASH_FLAG: BOOL := FALSE;

END_VAR
(*4.1.7.1.2*)
(*INIT AUT status lamp, this is used for Power up status,default status is F.W.E*)
IF	MODE_TRANSFER_FLAG = FALSE
THEN
	(*current status is F.W.E*)
	IF  AUX_EOT_STATUS = 3
	THEN
		INDICATOR_FWE_BRG := TRUE;
		INDICATOR_FWE_MCR := TRUE;
		INDICATOR_FWE_LC := TRUE;
	END_IF
END_IF

(*if current status is F.W.E, then after 30MIN, all indicator turn off and  AUT status is NONE, AUT_EOT_STATUS := 0*)
IF AUX_EOT_STATUS = 3
	AND MODE_TRANSFER_FLAG = FALSE
THEN
	TON_FWE_TIMER(IN := TRUE, PT := t#1800s);
ELSE
	(*if current status is not F.W.E,stop timer*)
	TON_FWE_TIMER(IN := FALSE, PT := t#1800s);
END_IF

(*F.W.E time out*)
IF  TON_FWE_TIMER.Q = TRUE
	AND  MODE_TRANSFER_FLAG = FALSE
THEN
	(*All the indicators should keep  OFF*)
	INDICATOR_STANDBY_BRG := FALSE;
	INDICATOR_STANDBY_MCR := FALSE;
	INDICATOR_STANDBY_LC := FALSE;

	INDICATOR_ATSEA_BRG := FALSE;
	INDICATOR_ATSEA_MCR := FALSE;
	INDICATOR_ATSEA_LC := FALSE;

	INDICATOR_FWE_BRG := FALSE;
	INDICATOR_FWE_MCR := FALSE;
	INDICATOR_FWE_LC := FALSE;

	(*change status to NONE*)
	AUX_EOT_STATUS := 0;
END_IF


(*generate flash pulse*)
INDICATOR_FLASH(ENABLE := TRUE, TIMELOW := t#0.5s, TIMEHIGH := t#0.5s);


(*********当前逻辑为standby确认需要MCR 按两次确认键才能成功转换, ATSEA 与 FWE 状态只需要按一次即可转换完成,当60秒未确认转换则该次转换取消,系统恢复之前状态***********)

				(*----------------------------standby logic----------------------------*)
(*standby button pressed from BRG and not during another switch process and current status is not STAND_BY*)
IF PUSHBUTTON_STANDBY_BRG = TRUE
	AND  MODE_TRANSFER_FLAG = FALSE
	 AND (AUX_EOT_STATUS <> 1)
THEN
	(*BRG pushbutton pressed flag set true, mode transfer set true, indicator flash  set true*)
	BRG_STANDBY_PRESSED_FLAG := TRUE;
	MODE_TRANSFER_FLAG := TRUE;
	STANDBY_PRO_IND_FLASH_FLAG := TRUE;

	(*The indicators of “STAND BY” both on BRG (PROEOT0002), MCR (PROEOT0018) and LC (PROEOT0034) will flash*)
	INDICATOR_STANDBY_BRG := INDICATOR_FLASH.OUT;
	INDICATOR_STANDBY_MCR := INDICATOR_FLASH.OUT;
	INDICATOR_STANDBY_LC := INDICATOR_FLASH.OUT;

	(*the EOT buzzers of BRG (PROEOT0015) and MCR (PROEOT0031) will be activated.*)
	BUZZER_BRG := TRUE;
	BUZZER_MCR := TRUE;

	(*start TIME OUT timer*)
	TON_TIMEOUT(IN := TRUE, PT := t#60s);
END_IF;

(*make  STANDBY INDICATOR keep FLASH*)
IF	STANDBY_PRO_IND_FLASH_FLAG = TRUE
THEN
	INDICATOR_STANDBY_BRG := INDICATOR_FLASH.OUT;
	INDICATOR_STANDBY_MCR := INDICATOR_FLASH.OUT;
	INDICATOR_STANDBY_LC := INDICATOR_FLASH.OUT;

	TON_TIMEOUT(IN := TRUE, PT := t#60s);
END_IF


(*The “STAND BY” pushbutton on MCR (PROEOT0017) is pressed first time*)
IF PUSHBUTTON_STANDBY_MCR = TRUE
THEN
	(* the “STAND BY” pushbutton on BRG is already pressed*)
	IF  BRG_STANDBY_PRESSED_FLAG = TRUE
		 AND  MCR_STANDBY_PRESSED_FLAG = FALSE
		 AND  MCR_STANDBY_FST_PRESSED_FLAG = FALSE
	THEN
		(*The buzzers of BRG and MCR will be silenced and the indicators still flashing*)
		BUZZER_BRG := FALSE;
		BUZZER_MCR := FALSE;

		(*MCR pushbutton pressed flag set true*)
		MCR_STANDBY_PRESSED_FLAG := TRUE;

		(*MCR pushbutton pressed first time flag set true*)
		MCR_STANDBY_FST_PRESSED_FLAG := TRUE;
	END_IF;
ELSE
	MCR_STANDBY_PRESSED_FLAG := FALSE;
END_IF


(*The “STAND BY” pushbutton on MCR (PROEOT0017) is pressed second time, that means the whole  transfer process completed*)
IF PUSHBUTTON_STANDBY_MCR = TRUE
	 AND MCR_STANDBY_PRESSED_FLAG = FALSE
	AND  MCR_STANDBY_FST_PRESSED_FLAG = TRUE
THEN
	(*All the “STAND BY” indicators should keep stable light*)
	INDICATOR_STANDBY_BRG := TRUE;
	INDICATOR_STANDBY_MCR := TRUE;
	INDICATOR_STANDBY_LC := TRUE;
	(*other indicators should keep light off*)
	INDICATOR_ATSEA_BRG := FALSE;
	INDICATOR_ATSEA_MCR := FALSE;
	INDICATOR_ATSEA_LC := FALSE;
	INDICATOR_FWE_BRG := FALSE;
	INDICATOR_FWE_MCR := FALSE;
	INDICATOR_FWE_LC := FALSE;
	(*current status set standby*)
	AUX_EOT_STATUS := 1;
	(* pushbutton pressed flag of MCR and BRG reset to FALSE*)
	MCR_STANDBY_PRESSED_FLAG := FALSE;
	BRG_STANDBY_PRESSED_FLAG := FALSE;
	MODE_TRANSFER_FLAG := FALSE;

	MCR_STANDBY_FST_PRESSED_FLAG := FALSE;
	MCR_ATSEA_FST_PRESSED_FLAG := FALSE;
	MCR_FWE_FST_PRESSED_FLAG := FALSE;

	(*indicator flash flag set false*)
	STANDBY_PRO_IND_FLASH_FLAG := FALSE;

	(*stop TIME OUT timer*)
	TON_TIMEOUT(IN := FALSE);
END_IF;

			(*----------------------------FWE logic----------------------------*)
(*F.W.E button pressed from BRG and not during another switch process and current status is not F.W.E*)
IF PUSHBUTTON_FWE_BRG = TRUE
	 AND MODE_TRANSFER_FLAG = FALSE
	 AND (AUX_EOT_STATUS <> 3)
THEN
	(*The indicators of F.W.E” both on BRG, MCR and LC will flash*)
	INDICATOR_FWE_BRG := INDICATOR_FLASH.OUT;;
	INDICATOR_FWE_MCR := INDICATOR_FLASH.OUT;;
	INDICATOR_FWE_LC := INDICATOR_FLASH.OUT;;

	(*the EOT buzzers of BRG and MCR will be activated.*)
	BUZZER_BRG := TRUE;
	BUZZER_MCR := TRUE;

	(*BRG pushbutton pressed flag set true, mode transfer set true, indicator flash flag set true*)
	BRG_FWE_PRESSED_FLAG := TRUE;
	MODE_TRANSFER_FLAG := TRUE;
	FWE_PRO_IND_FLASH_FLAG := TRUE;

	(*start TIME OUT timer*)
	TON_TIMEOUT(IN := TRUE, PT := t#60s);
END_IF;


(*make  FWE PROCESS  INDICATOR keep FLASH*)
IF	FWE_PRO_IND_FLASH_FLAG = TRUE
THEN
	INDICATOR_FWE_BRG := INDICATOR_FLASH.OUT;
	INDICATOR_FWE_MCR := INDICATOR_FLASH.OUT;
	INDICATOR_FWE_LC := INDICATOR_FLASH.OUT;

	TON_TIMEOUT(IN := TRUE, PT := t#60s);
END_IF

(*The “F.W.E” pushbutton on MCR is pressed first time*)
IF PUSHBUTTON_FWE_MCR
THEN
	(* the “F.W.E” pushbutton on BRG is already pressed*)
	IF  BRG_FWE_PRESSED_FLAG = TRUE
	 AND MCR_FWE_PRESSED_FLAG = FALSE
	THEN
		(*The buzzers of BRG and MCR will be silenced and the indicators still flashing*)
		BUZZER_BRG := FALSE;
		BUZZER_MCR := FALSE;

		(*MCR pushbutton pressed flag set true*)
		MCR_FWE_PRESSED_FLAG := TRUE;
	END_IF;
END_IF;

(*The “F.W.E” pushbutton on MCR is pressed second time, that means the hole mode transfer process completed*)
IF PUSHBUTTON_FWE_MCR = TRUE
	 AND MCR_FWE_PRESSED_FLAG = TRUE
THEN
	(*All the “F.W.E” indicators should keep stable light*)
	INDICATOR_FWE_BRG := TRUE;
	INDICATOR_FWE_MCR := TRUE;
	INDICATOR_FWE_LC := TRUE;
	(*other indicators should keep light off*)
	INDICATOR_ATSEA_BRG := FALSE;
	INDICATOR_ATSEA_MCR := FALSE;
	INDICATOR_ATSEA_LC := FALSE;
	INDICATOR_STANDBY_BRG := FALSE;
	INDICATOR_STANDBY_MCR := FALSE;
	INDICATOR_STANDBY_LC := FALSE;
	(*current status set F.W.E*)
	AUX_EOT_STATUS := 3;
	(* pushbutton pressed flag of MCR and BRG reset to FALSE*)
	MCR_FWE_PRESSED_FLAG := FALSE;
	BRG_FWE_PRESSED_FLAG := FALSE;
	MODE_TRANSFER_FLAG := FALSE;

	(*set FWE PROCESS indicator flash flag false*)
	FWE_PRO_IND_FLASH_FLAG := FALSE;

	(*stop TIME OUT timer*)
	TON_TIMEOUT(IN := FALSE);
END_IF;


			(*----------------------------ATSEA  logic----------------------------*)
(*ATSEA button pressed from BRG and not during another switch process and current status is not ATSEA and not F.W.E*)
IF PUSHBUTTON_ATSEA_BRG = TRUE
	AND MODE_TRANSFER_FLAG = FALSE
	AND (AUX_EOT_STATUS <> 3)
	AND (AUX_EOT_STATUS <> 2)
THEN
	(*The indicators of 'ATSEA” both on BRG, MCR and LC will flash*)
	INDICATOR_ATSEA_BRG := INDICATOR_FLASH.OUT;
	INDICATOR_ATSEA_MCR := INDICATOR_FLASH.OUT;
	INDICATOR_ATSEA_LC := INDICATOR_FLASH.OUT;

	(*the EOT buzzers of BRG and MCR will be activated.*)
	BUZZER_BRG := TRUE;
	BUZZER_MCR := TRUE;

	(*BRG pushbutton pressed flag set true, mode transfer set true*)
	BRG_ATSEA_PRESSED_FLAG := TRUE;
	MODE_TRANSFER_FLAG := TRUE;

	(*ATSEA process indicator flash flag*)
	ATSEA_PRO_IND_FLASH_FLAG := TRUE;

	(*start TIME OUT timer*)
	TON_TIMEOUT(IN := TRUE, PT := t#60s);
END_IF;


(*make ATSEA PROCESS indicator keep flash*)
IF	ATSEA_PRO_IND_FLASH_FLAG = TRUE
THEN
	INDICATOR_ATSEA_BRG := INDICATOR_FLASH.OUT;
	INDICATOR_ATSEA_MCR := INDICATOR_FLASH.OUT;
	INDICATOR_ATSEA_LC := INDICATOR_FLASH.OUT;

	TON_TIMEOUT(IN := TRUE, PT := t#60s);
END_IF

(*The “ATSEA” pushbutton on MCR is pressed first time*)
IF PUSHBUTTON_ATSEA_MCR
THEN
	(* the “ATSEA” pushbutton on BRG is already pressed*)
	IF  BRG_ATSEA_PRESSED_FLAG = TRUE
	 AND MCR_ATSEA_PRESSED_FLAG = FALSE
	THEN
		(*The buzzers of BRG and MCR will be silenced and the indicators still flashing*)
		BUZZER_BRG := FALSE;
		BUZZER_MCR := FALSE;

		(*MCR pushbutton pressed flag set true*)
		MCR_ATSEA_PRESSED_FLAG := TRUE;
	END_IF;
END_IF;

(*The “ATSEA” pushbutton on MCR is pressed second time, that means the hole mode transfer process completed*)
IF PUSHBUTTON_ATSEA_MCR = TRUE
	 AND MCR_ATSEA_PRESSED_FLAG = TRUE
THEN
	(*All the “ATSEA” indicators should keep stable light*)
	INDICATOR_ATSEA_BRG := TRUE;
	INDICATOR_ATSEA_MCR := TRUE;
	INDICATOR_ATSEA_LC := TRUE;
	(*other indicators should keep light off*)
	INDICATOR_FWE_BRG := FALSE;
	INDICATOR_FWE_MCR := FALSE;
	INDICATOR_FWE_LC := FALSE;
	INDICATOR_STANDBY_BRG := FALSE;
	INDICATOR_STANDBY_MCR := FALSE;
	INDICATOR_STANDBY_LC := FALSE;
	(*current status set ATSEA*)
	AUX_EOT_STATUS := 2;
	(* pushbutton pressed flag of MCR and BRG reset to FALSE*)
	MCR_ATSEA_PRESSED_FLAG := FALSE;
	BRG_ATSEA_PRESSED_FLAG := FALSE;
	MODE_TRANSFER_FLAG := FALSE;

	(*ATSEA  PROCESS indicator flash flag set false*)
	ATSEA_PRO_IND_FLASH_FLAG := FALSE;

	(*start TIME OUT timer*)
	TON_TIMEOUT(IN := FALSE);
END_IF;

(*TIME OUT PROCESS*)
IF  TON_TIMEOUT.Q = TRUE
	AND  MODE_TRANSFER_FLAG = TRUE
THEN
	(*RESET  transfer process*)
	(*all the flag set false*)
	MODE_TRANSFER_FLAG := FALSE;

	BRG_STANDBY_PRESSED_FLAG := FALSE;
	MCR_STANDBY_PRESSED_FLAG := FALSE;

	BRG_ATSEA_PRESSED_FLAG := FALSE;
	MCR_ATSEA_PRESSED_FLAG := FALSE;

	BRG_FWE_PRESSED_FLAG := FALSE;
	MCR_FWE_PRESSED_FLAG := FALSE;

	MCR_STANDBY_FST_PRESSED_FLAG := FALSE;
	MCR_ATSEA_FST_PRESSED_FLAG := FALSE;
	MCR_FWE_FST_PRESSED_FLAG := FALSE;

	(*indicator flash flag*)
	STANDBY_PRO_IND_FLASH_FLAG := FALSE;
	ATSEA_PRO_IND_FLASH_FLAG := FALSE;
	FWE_PRO_IND_FLASH_FLAG := FALSE;

	(*all buzzers turned off*)
	BUZZER_BRG := FALSE;
	BUZZER_MCR := FALSE;

	(*STOP TIMEOUT timer*)
	TON_TIMEOUT(IN := FALSE);

	(*current status is none*)
	IF AUX_EOT_STATUS = 0
	THEN
		(*All the indicators should keep  OFF*)
		INDICATOR_STANDBY_BRG := FALSE;
		INDICATOR_STANDBY_MCR := FALSE;
		INDICATOR_STANDBY_LC := FALSE;

		INDICATOR_ATSEA_BRG := FALSE;
		INDICATOR_ATSEA_MCR := FALSE;
		INDICATOR_ATSEA_LC := FALSE;
	
